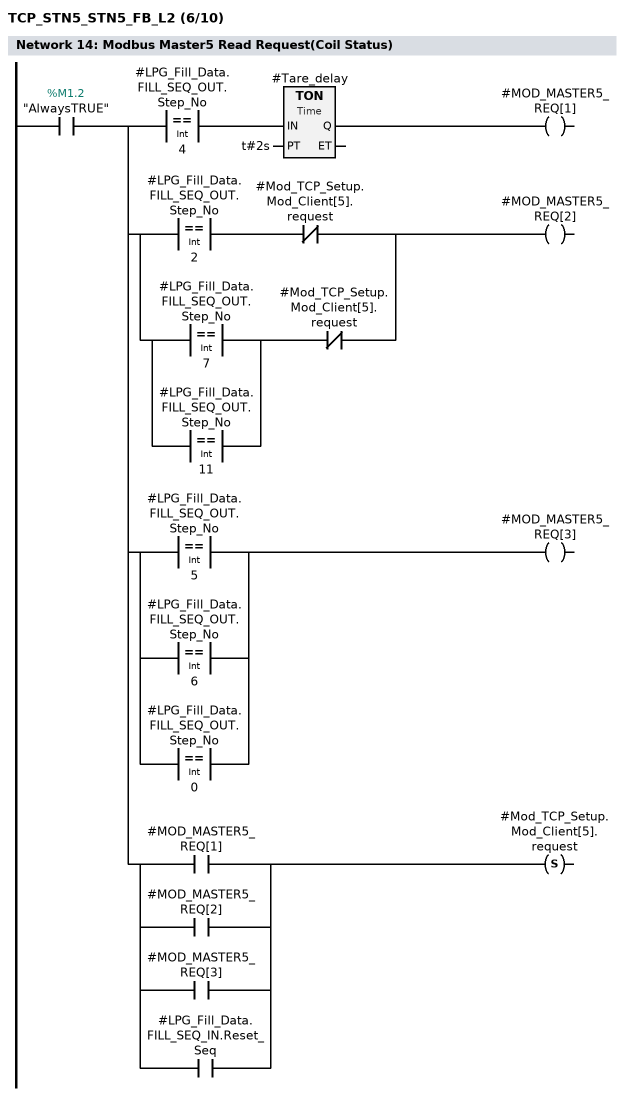
   RUNG wire#powerrail
      Contact( "AlwaysTRUE" )
      wire#w1
      { S7_Templates := "SrcType := Int" } EQ_Contact(in1 := #LPG_Fill_Data.FILL_SEQ_OUT.Step_No, in2 := 4)
      { S7_Templates := "time_type := Time" } #Tare_delay.TON(pt := t#2s, et =>)
      Coil( #MOD_MASTER5_REQ[1] )
   END_RUNG
   RUNG wire#w1
      { S7_Templates := "SrcType := Int" } EQ_Contact(in1 := #LPG_Fill_Data.FILL_SEQ_OUT.Step_No, in2 := 2)
      I_Contact( #Mod_TCP_Setup.Mod_Client[5].request )
      wire#w2
      Coil( #MOD_MASTER5_REQ[2] )
   END_RUNG
   RUNG wire#w1
      { S7_Templates := "SrcType := Int" } EQ_Contact(in1 := #LPG_Fill_Data.FILL_SEQ_OUT.Step_No, in2 := 7)
      wire#w3
      I_Contact( #Mod_TCP_Setup.Mod_Client[5].request )
   END_RUNG wire#w2
   RUNG wire#w1
      { S7_Templates := "SrcType := Int" } EQ_Contact(in1 := #LPG_Fill_Data.FILL_SEQ_OUT.Step_No, in2 := 11)
   END_RUNG wire#w3
   RUNG wire#w1
      { S7_Templates := "SrcType := Int" } EQ_Contact(in1 := #LPG_Fill_Data.FILL_SEQ_OUT.Step_No, in2 := 5)
      wire#w4
      Coil( #MOD_MASTER5_REQ[3] )
   END_RUNG
   RUNG wire#w1
      { S7_Templates := "SrcType := Int" } EQ_Contact(in1 := #LPG_Fill_Data.FILL_SEQ_OUT.Step_No, in2 := 6)
   END_RUNG wire#w4
   RUNG wire#w1
      { S7_Templates := "SrcType := Int" } EQ_Contact(in1 := #LPG_Fill_Data.FILL_SEQ_OUT.Step_No, in2 := 0)
   END_RUNG wire#w4
   RUNG wire#w1
      Contact( #MOD_MASTER5_REQ[1] )
      wire#w5
      S_Coil( #Mod_TCP_Setup.Mod_Client[5].request )
   END_RUNG
   RUNG wire#w1
      Contact( #MOD_MASTER5_REQ[2] )
   END_RUNG wire#w5
   RUNG wire#w1
      Contact( #MOD_MASTER5_REQ[3] )
   END_RUNG wire#w5
   RUNG wire#w1
      Contact( #LPG_Fill_Data.FILL_SEQ_IN.Reset_Seq )
   END_RUNG wire#w5
   // the same network as SCL:
   #Tare_delay(IN := "AlwaysTRUE" AND (#LPG_Fill_Data.FILL_SEQ_OUT.Step_No = 4), PT := t#2s);   // TON
   #MOD_MASTER5_REQ[1] := #Tare_delay.Q;
   #MOD_MASTER5_REQ[2] := "AlwaysTRUE" AND (((#LPG_Fill_Data.FILL_SEQ_OUT.Step_No = 2) AND NOT #Mod_TCP_Setup.Mod_Client[5].request) OR (((#LPG_Fill_Data.FILL_SEQ_OUT.Step_No = 7) OR (#LPG_Fill_Data.FILL_SEQ_OUT.Step_No = 11)) AND NOT #Mod_TCP_Setup.Mod_Client[5].request));
   #MOD_MASTER5_REQ[3] := "AlwaysTRUE" AND ((#LPG_Fill_Data.FILL_SEQ_OUT.Step_No = 5) OR (#LPG_Fill_Data.FILL_SEQ_OUT.Step_No = 6) OR (#LPG_Fill_Data.FILL_SEQ_OUT.Step_No = 0));
   IF "AlwaysTRUE" AND (#MOD_MASTER5_REQ[1] OR #MOD_MASTER5_REQ[2] OR #MOD_MASTER5_REQ[3] OR #LPG_Fill_Data.FILL_SEQ_IN.Reset_Seq) THEN
       #Mod_TCP_Setup.Mod_Client[5].request := TRUE;
   END_IF;
END_REGION

REGION Network 15: Modbus Master5 Read Coil Status
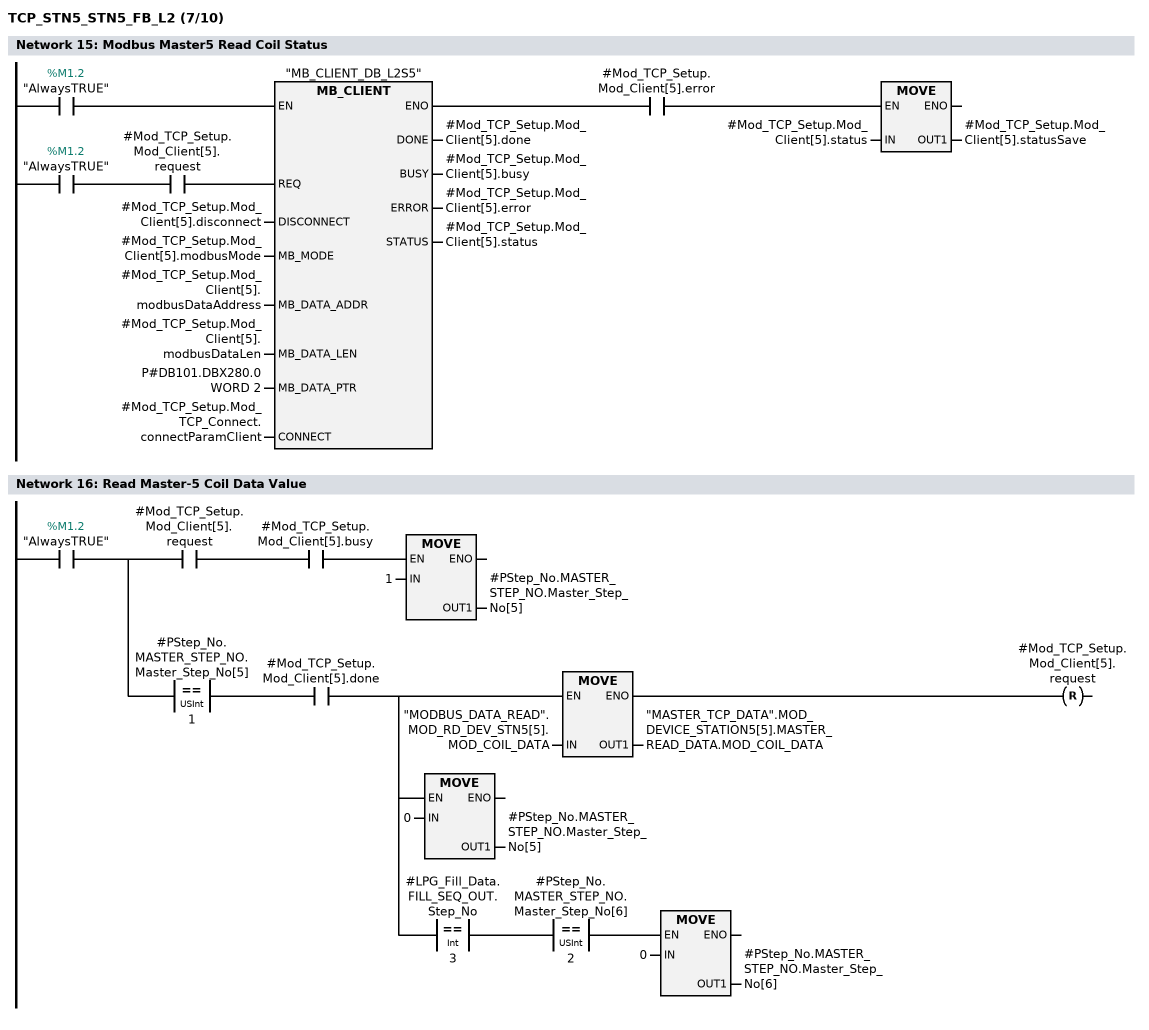
   RUNG wire#powerrail
      Contact( "AlwaysTRUE" )
      "MB_CLIENT_DB_L2S5".MB_CLIENT(REQ := wire#w1, DISCONNECT := #Mod_TCP_Setup.Mod_Client[5].disconnect, MB_MODE := #Mod_TCP_Setup.Mod_Client[5].modbusMode, MB_DATA_ADDR := #Mod_TCP_Setup.Mod_Client[5].modbusDataAddress, MB_DATA_LEN := #Mod_TCP_Setup.Mod_Client[5].modbusDataLen, MB_DATA_PTR := P#DB101.DBX280.0 WORD 2, CONNECT := #Mod_TCP_Setup.Mod_TCP_Connect.connectParamClient, DONE => #Mod_TCP_Setup.Mod_Client[5].done, BUSY => #Mod_TCP_Setup.Mod_Client[5].busy, ERROR => #Mod_TCP_Setup.Mod_Client[5].error, STATUS => #Mod_TCP_Setup.Mod_Client[5].status)
      Contact( #Mod_TCP_Setup.Mod_Client[5].error )
      Move(in := #Mod_TCP_Setup.Mod_Client[5].status, out1 => #Mod_TCP_Setup.Mod_Client[5].statusSave)
   END_RUNG
   RUNG wire#powerrail
      Contact( "AlwaysTRUE" )
      Contact( #Mod_TCP_Setup.Mod_Client[5].request )
   END_RUNG wire#w1
   // the same network as SCL:
   "MB_CLIENT_DB_L2S5"(EN := "AlwaysTRUE",   // MB_CLIENT
                       REQ := "AlwaysTRUE" AND #Mod_TCP_Setup.Mod_Client[5].request,
                       DISCONNECT := #Mod_TCP_Setup.Mod_Client[5].disconnect,
                       MB_MODE := #Mod_TCP_Setup.Mod_Client[5].modbusMode,
                       MB_DATA_ADDR := #Mod_TCP_Setup.Mod_Client[5].modbusDataAddress,
                       MB_DATA_LEN := #Mod_TCP_Setup.Mod_Client[5].modbusDataLen,
                       MB_DATA_PTR := P#DB101.DBX280.0 WORD 2,
                       CONNECT := #Mod_TCP_Setup.Mod_TCP_Connect.connectParamClient,
                       DONE => #Mod_TCP_Setup.Mod_Client[5].done,
                       BUSY => #Mod_TCP_Setup.Mod_Client[5].busy,
                       ERROR => #Mod_TCP_Setup.Mod_Client[5].error,
                       STATUS => #Mod_TCP_Setup.Mod_Client[5].status,
                       ENO => #_w1);
   IF #_w1 AND #Mod_TCP_Setup.Mod_Client[5].error THEN
       #Mod_TCP_Setup.Mod_Client[5].statusSave := #Mod_TCP_Setup.Mod_Client[5].status;
   END_IF;
END_REGION

REGION Network 16: Read Master-5 Coil Data Value
   RUNG wire#powerrail
      Contact( "AlwaysTRUE" )
      wire#w1
      Contact( #Mod_TCP_Setup.Mod_Client[5].request )
      Contact( #Mod_TCP_Setup.Mod_Client[5].busy )
      Move(in := 1, out1 => #PStep_No.MASTER_STEP_NO.Master_Step_No[5])
   END_RUNG
   RUNG wire#w1
      { S7_Templates := "SrcType := USInt" } EQ_Contact(in1 := #PStep_No.MASTER_STEP_NO.Master_Step_No[5], in2 := 1)
      Contact( #Mod_TCP_Setup.Mod_Client[5].done )
      wire#w2
      Move(in := "MODBUS_DATA_READ".MOD_RD_DEV_STN5[5].MOD_COIL_DATA, out1 => "MASTER_TCP_DATA".MOD_DEVICE_STATION5[5].MASTER_READ_DATA.MOD_COIL_DATA)
      R_Coil( #Mod_TCP_Setup.Mod_Client[5].request )
   END_RUNG
   RUNG wire#w2
      Move(in := 0, out1 => #PStep_No.MASTER_STEP_NO.Master_Step_No[5])
   END_RUNG
   RUNG wire#w2
      { S7_Templates := "SrcType := Int" } EQ_Contact(in1 := #LPG_Fill_Data.FILL_SEQ_OUT.Step_No, in2 := 3)
      { S7_Templates := "SrcType := USInt" } EQ_Contact(in1 := #PStep_No.MASTER_STEP_NO.Master_Step_No[6], in2 := 2)
      Move(in := 0, out1 => #PStep_No.MASTER_STEP_NO.Master_Step_No[6])
   END_RUNG
   // the same network as SCL:
   IF "AlwaysTRUE" AND #Mod_TCP_Setup.Mod_Client[5].request AND #Mod_TCP_Setup.Mod_Client[5].busy THEN
       #PStep_No.MASTER_STEP_NO.Master_Step_No[5] := 1;
   END_IF;
   #_w1 := "AlwaysTRUE" AND (#PStep_No.MASTER_STEP_NO.Master_Step_No[5] = 1) AND #Mod_TCP_Setup.Mod_Client[5].done;
   IF #_w1 THEN
       "MASTER_TCP_DATA".MOD_DEVICE_STATION5[5].MASTER_READ_DATA.MOD_COIL_DATA := "MODBUS_DATA_READ".MOD_RD_DEV_STN5[5].MOD_COIL_DATA;
       #Mod_TCP_Setup.Mod_Client[5].request := FALSE;
       #PStep_No.MASTER_STEP_NO.Master_Step_No[5] := 0;
   END_IF;
   IF #_w1 AND (#LPG_Fill_Data.FILL_SEQ_OUT.Step_No = 3) AND (#PStep_No.MASTER_STEP_NO.Master_Step_No[6] = 2) THEN
       #PStep_No.MASTER_STEP_NO.Master_Step_No[6] := 0;
   END_IF;
END_REGION

REGION Network 17: Write Coil Data
   // if multiple bit write not working
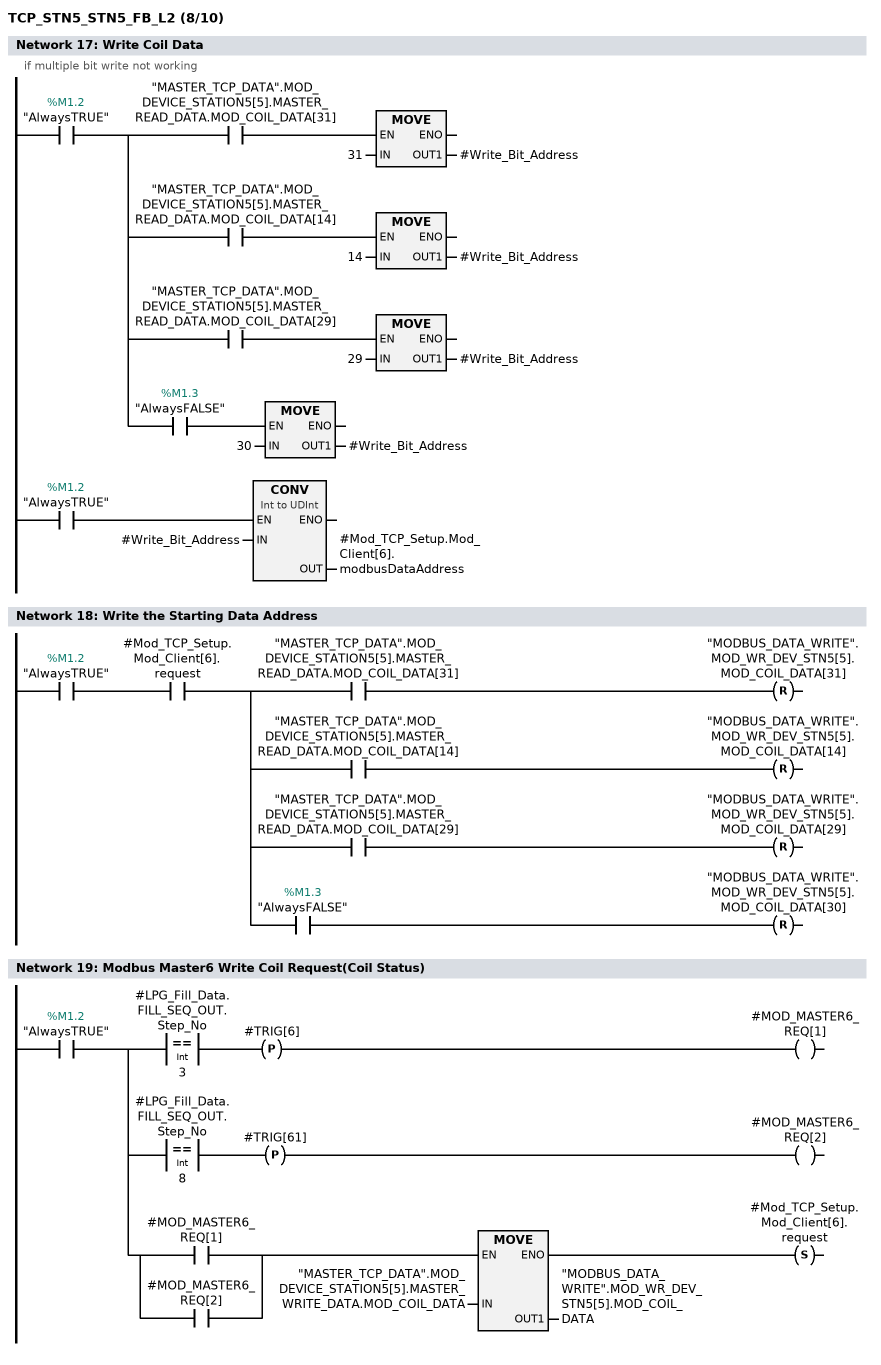
   RUNG wire#powerrail
      Contact( "AlwaysTRUE" )
      wire#w1
      Contact( "MASTER_TCP_DATA".MOD_DEVICE_STATION5[5].MASTER_READ_DATA.MOD_COIL_DATA[31] )
      Move(in := 31, out1 => #Write_Bit_Address)
   END_RUNG
   RUNG wire#w1
      Contact( "MASTER_TCP_DATA".MOD_DEVICE_STATION5[5].MASTER_READ_DATA.MOD_COIL_DATA[14] )
      Move(in := 14, out1 => #Write_Bit_Address)
   END_RUNG
   RUNG wire#w1
      Contact( "MASTER_TCP_DATA".MOD_DEVICE_STATION5[5].MASTER_READ_DATA.MOD_COIL_DATA[29] )
      Move(in := 29, out1 => #Write_Bit_Address)
   END_RUNG
   RUNG wire#w1
      Contact( "AlwaysFALSE" )
      Move(in := 30, out1 => #Write_Bit_Address)
   END_RUNG
   RUNG wire#powerrail
      Contact( "AlwaysTRUE" )
      { S7_Templates := "[SrcType := Int, DestType := UDInt]" } Convert(in := #Write_Bit_Address, out => #Mod_TCP_Setup.Mod_Client[6].modbusDataAddress)
   END_RUNG
   // the same network as SCL:
   IF "AlwaysTRUE" AND "MASTER_TCP_DATA".MOD_DEVICE_STATION5[5].MASTER_READ_DATA.MOD_COIL_DATA[31] THEN
       #Write_Bit_Address := 31;
   END_IF;
   IF "AlwaysTRUE" AND "MASTER_TCP_DATA".MOD_DEVICE_STATION5[5].MASTER_READ_DATA.MOD_COIL_DATA[14] THEN
       #Write_Bit_Address := 14;
   END_IF;
   IF "AlwaysTRUE" AND "MASTER_TCP_DATA".MOD_DEVICE_STATION5[5].MASTER_READ_DATA.MOD_COIL_DATA[29] THEN
       #Write_Bit_Address := 29;
   END_IF;
   IF "AlwaysTRUE" AND "AlwaysFALSE" THEN #Write_Bit_Address := 30; END_IF;
   IF "AlwaysTRUE" THEN
       #Mod_TCP_Setup.Mod_Client[6].modbusDataAddress := INT_TO_UDINT(#Write_Bit_Address);
   END_IF;
END_REGION

REGION Network 18: Write the Starting Data Address
   RUNG wire#powerrail
      Contact( "AlwaysTRUE" )
      Contact( #Mod_TCP_Setup.Mod_Client[6].request )
      wire#w1
      Contact( "MASTER_TCP_DATA".MOD_DEVICE_STATION5[5].MASTER_READ_DATA.MOD_COIL_DATA[31] )
      R_Coil( "MODBUS_DATA_WRITE".MOD_WR_DEV_STN5[5].MOD_COIL_DATA[31] )
   END_RUNG
   RUNG wire#w1
      Contact( "MASTER_TCP_DATA".MOD_DEVICE_STATION5[5].MASTER_READ_DATA.MOD_COIL_DATA[14] )
      R_Coil( "MODBUS_DATA_WRITE".MOD_WR_DEV_STN5[5].MOD_COIL_DATA[14] )
   END_RUNG
   RUNG wire#w1
      Contact( "MASTER_TCP_DATA".MOD_DEVICE_STATION5[5].MASTER_READ_DATA.MOD_COIL_DATA[29] )
      R_Coil( "MODBUS_DATA_WRITE".MOD_WR_DEV_STN5[5].MOD_COIL_DATA[29] )
   END_RUNG
   RUNG wire#w1
      Contact( "AlwaysFALSE" )
      R_Coil( "MODBUS_DATA_WRITE".MOD_WR_DEV_STN5[5].MOD_COIL_DATA[30] )
   END_RUNG
   // the same network as SCL:
   #_w1 := "AlwaysTRUE" AND #Mod_TCP_Setup.Mod_Client[6].request;
   IF #_w1 AND "MASTER_TCP_DATA".MOD_DEVICE_STATION5[5].MASTER_READ_DATA.MOD_COIL_DATA[31] THEN
       "MODBUS_DATA_WRITE".MOD_WR_DEV_STN5[5].MOD_COIL_DATA[31] := FALSE;
   END_IF;
   IF #_w1 AND "MASTER_TCP_DATA".MOD_DEVICE_STATION5[5].MASTER_READ_DATA.MOD_COIL_DATA[14] THEN
       "MODBUS_DATA_WRITE".MOD_WR_DEV_STN5[5].MOD_COIL_DATA[14] := FALSE;
   END_IF;
   IF #_w1 AND "MASTER_TCP_DATA".MOD_DEVICE_STATION5[5].MASTER_READ_DATA.MOD_COIL_DATA[29] THEN
       "MODBUS_DATA_WRITE".MOD_WR_DEV_STN5[5].MOD_COIL_DATA[29] := FALSE;
   END_IF;
   IF #_w1 AND "AlwaysFALSE" THEN "MODBUS_DATA_WRITE".MOD_WR_DEV_STN5[5].MOD_COIL_DATA[30] := FALSE; END_IF;
END_REGION

REGION Network 19: Modbus Master6 Write Coil Request(Coil Status)
   RUNG wire#powerrail
      Contact( "AlwaysTRUE" )
      wire#w1
      { S7_Templates := "SrcType := Int" } EQ_Contact(in1 := #LPG_Fill_Data.FILL_SEQ_OUT.Step_No, in2 := 3)
      P_Trig( #TRIG[6] )
      Coil( #MOD_MASTER6_REQ[1] )
   END_RUNG
   RUNG wire#w1
      { S7_Templates := "SrcType := Int" } EQ_Contact(in1 := #LPG_Fill_Data.FILL_SEQ_OUT.Step_No, in2 := 8)
      P_Trig( #TRIG[61] )
      Coil( #MOD_MASTER6_REQ[2] )
   END_RUNG
   RUNG wire#w1
      Contact( #MOD_MASTER6_REQ[1] )
      wire#w2
      Move(in := "MASTER_TCP_DATA".MOD_DEVICE_STATION5[5].MASTER_WRITE_DATA.MOD_COIL_DATA, out1 => "MODBUS_DATA_WRITE".MOD_WR_DEV_STN5[5].MOD_COIL_DATA)
      S_Coil( #Mod_TCP_Setup.Mod_Client[6].request )
   END_RUNG
   RUNG wire#w1
      Contact( #MOD_MASTER6_REQ[2] )
   END_RUNG wire#w2
   // the same network as SCL:
   #_w1 := "AlwaysTRUE" AND (#LPG_Fill_Data.FILL_SEQ_OUT.Step_No = 3);
   #_w2 := #_w1 AND NOT #TRIG[6];   // rising edge
   #TRIG[6] := #_w1;
   #MOD_MASTER6_REQ[1] := #_w2;
   #_w3 := "AlwaysTRUE" AND (#LPG_Fill_Data.FILL_SEQ_OUT.Step_No = 8);
   #_w4 := #_w3 AND NOT #TRIG[61];   // rising edge
   #TRIG[61] := #_w3;
   #MOD_MASTER6_REQ[2] := #_w4;
   IF "AlwaysTRUE" AND (#MOD_MASTER6_REQ[1] OR #MOD_MASTER6_REQ[2]) THEN
       "MODBUS_DATA_WRITE".MOD_WR_DEV_STN5[5].MOD_COIL_DATA := "MASTER_TCP_DATA".MOD_DEVICE_STATION5[5].MASTER_WRITE_DATA.MOD_COIL_DATA;
       #Mod_TCP_Setup.Mod_Client[6].request := TRUE;
   END_IF;
END_REGION

REGION Network 20: Modbus Master6 Write Coil Status
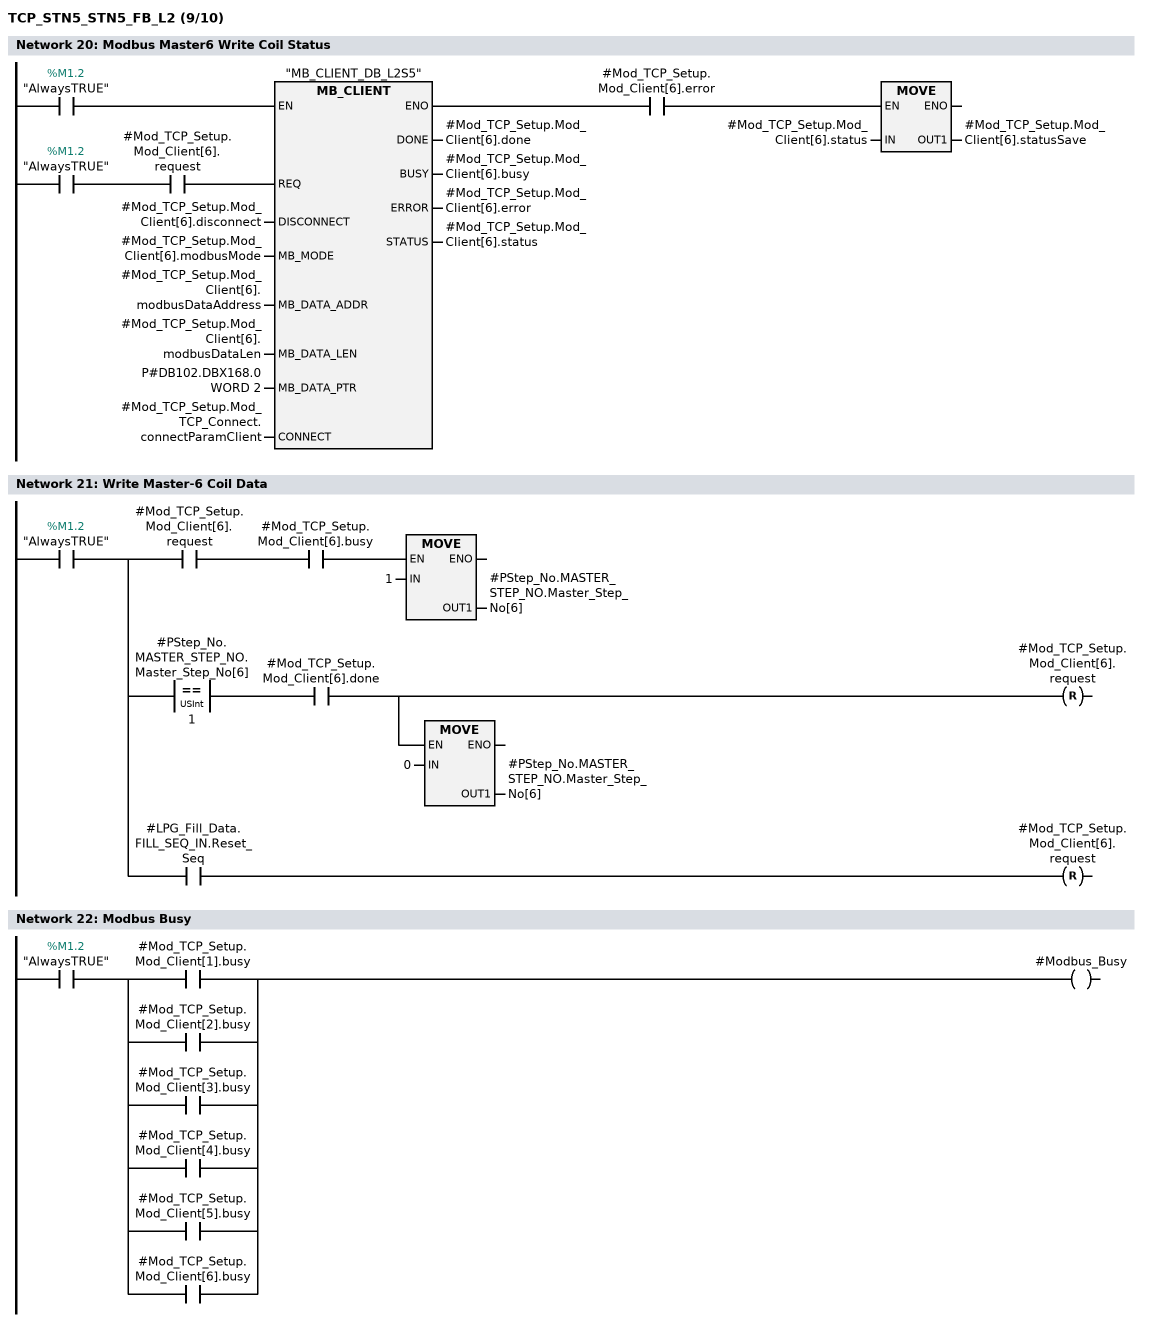
   RUNG wire#powerrail
      Contact( "AlwaysTRUE" )
      "MB_CLIENT_DB_L2S5".MB_CLIENT(REQ := wire#w1, DISCONNECT := #Mod_TCP_Setup.Mod_Client[6].disconnect, MB_MODE := #Mod_TCP_Setup.Mod_Client[6].modbusMode, MB_DATA_ADDR := #Mod_TCP_Setup.Mod_Client[6].modbusDataAddress, MB_DATA_LEN := #Mod_TCP_Setup.Mod_Client[6].modbusDataLen, MB_DATA_PTR := P#DB102.DBX168.0 WORD 2, CONNECT := #Mod_TCP_Setup.Mod_TCP_Connect.connectParamClient, DONE => #Mod_TCP_Setup.Mod_Client[6].done, BUSY => #Mod_TCP_Setup.Mod_Client[6].busy, ERROR => #Mod_TCP_Setup.Mod_Client[6].error, STATUS => #Mod_TCP_Setup.Mod_Client[6].status)
      Contact( #Mod_TCP_Setup.Mod_Client[6].error )
      Move(in := #Mod_TCP_Setup.Mod_Client[6].status, out1 => #Mod_TCP_Setup.Mod_Client[6].statusSave)
   END_RUNG
   RUNG wire#powerrail
      Contact( "AlwaysTRUE" )
      Contact( #Mod_TCP_Setup.Mod_Client[6].request )
   END_RUNG wire#w1
   // the same network as SCL:
   "MB_CLIENT_DB_L2S5"(EN := "AlwaysTRUE",   // MB_CLIENT
                       REQ := "AlwaysTRUE" AND #Mod_TCP_Setup.Mod_Client[6].request,
                       DISCONNECT := #Mod_TCP_Setup.Mod_Client[6].disconnect,
                       MB_MODE := #Mod_TCP_Setup.Mod_Client[6].modbusMode,
                       MB_DATA_ADDR := #Mod_TCP_Setup.Mod_Client[6].modbusDataAddress,
                       MB_DATA_LEN := #Mod_TCP_Setup.Mod_Client[6].modbusDataLen,
                       MB_DATA_PTR := P#DB102.DBX168.0 WORD 2,
                       CONNECT := #Mod_TCP_Setup.Mod_TCP_Connect.connectParamClient,
                       DONE => #Mod_TCP_Setup.Mod_Client[6].done,
                       BUSY => #Mod_TCP_Setup.Mod_Client[6].busy,
                       ERROR => #Mod_TCP_Setup.Mod_Client[6].error,
                       STATUS => #Mod_TCP_Setup.Mod_Client[6].status,
                       ENO => #_w1);
   IF #_w1 AND #Mod_TCP_Setup.Mod_Client[6].error THEN
       #Mod_TCP_Setup.Mod_Client[6].statusSave := #Mod_TCP_Setup.Mod_Client[6].status;
   END_IF;
END_REGION

REGION Network 21: Write Master-6 Coil Data
   RUNG wire#powerrail
      Contact( "AlwaysTRUE" )
      wire#w1
      Contact( #Mod_TCP_Setup.Mod_Client[6].request )
      Contact( #Mod_TCP_Setup.Mod_Client[6].busy )
      Move(in := 1, out1 => #PStep_No.MASTER_STEP_NO.Master_Step_No[6])
   END_RUNG
   RUNG wire#w1
      { S7_Templates := "SrcType := USInt" } EQ_Contact(in1 := #PStep_No.MASTER_STEP_NO.Master_Step_No[6], in2 := 1)
      Contact( #Mod_TCP_Setup.Mod_Client[6].done )
      wire#w2
      R_Coil( #Mod_TCP_Setup.Mod_Client[6].request )
   END_RUNG
   RUNG wire#w2
      Move(in := 0, out1 => #PStep_No.MASTER_STEP_NO.Master_Step_No[6])
   END_RUNG
   RUNG wire#w1
      Contact( #LPG_Fill_Data.FILL_SEQ_IN.Reset_Seq )
      R_Coil( #Mod_TCP_Setup.Mod_Client[6].request )
   END_RUNG
   // the same network as SCL:
   IF "AlwaysTRUE" AND #Mod_TCP_Setup.Mod_Client[6].request AND #Mod_TCP_Setup.Mod_Client[6].busy THEN
       #PStep_No.MASTER_STEP_NO.Master_Step_No[6] := 1;
   END_IF;
   #_w1 := "AlwaysTRUE" AND (#PStep_No.MASTER_STEP_NO.Master_Step_No[6] = 1) AND #Mod_TCP_Setup.Mod_Client[6].done;
   IF #_w1 THEN
       #Mod_TCP_Setup.Mod_Client[6].request := FALSE;
       #PStep_No.MASTER_STEP_NO.Master_Step_No[6] := 0;
   END_IF;
   IF "AlwaysTRUE" AND #LPG_Fill_Data.FILL_SEQ_IN.Reset_Seq THEN
       #Mod_TCP_Setup.Mod_Client[6].request := FALSE;
   END_IF;
END_REGION

REGION Network 22: Modbus Busy
   RUNG wire#powerrail
      Contact( "AlwaysTRUE" )
      wire#w1
      Contact( #Mod_TCP_Setup.Mod_Client[1].busy )
      wire#w2
      Coil( #Modbus_Busy )
   END_RUNG
   RUNG wire#w1
      Contact( #Mod_TCP_Setup.Mod_Client[2].busy )
   END_RUNG wire#w2
   RUNG wire#w1
      Contact( #Mod_TCP_Setup.Mod_Client[3].busy )
   END_RUNG wire#w2
   RUNG wire#w1
      Contact( #Mod_TCP_Setup.Mod_Client[4].busy )
   END_RUNG wire#w2
   RUNG wire#w1
      Contact( #Mod_TCP_Setup.Mod_Client[5].busy )
   END_RUNG wire#w2
   RUNG wire#w1
      Contact( #Mod_TCP_Setup.Mod_Client[6].busy )
   END_RUNG wire#w2
   // the same network as SCL:
   #Modbus_Busy := "AlwaysTRUE" AND (#Mod_TCP_Setup.Mod_Client[1].busy OR #Mod_TCP_Setup.Mod_Client[2].busy OR #Mod_TCP_Setup.Mod_Client[3].busy OR #Mod_TCP_Setup.Mod_Client[4].busy OR #Mod_TCP_Setup.Mod_Client[5].busy OR #Mod_TCP_Setup.Mod_Client[6].busy);
END_REGION

REGION Network 23
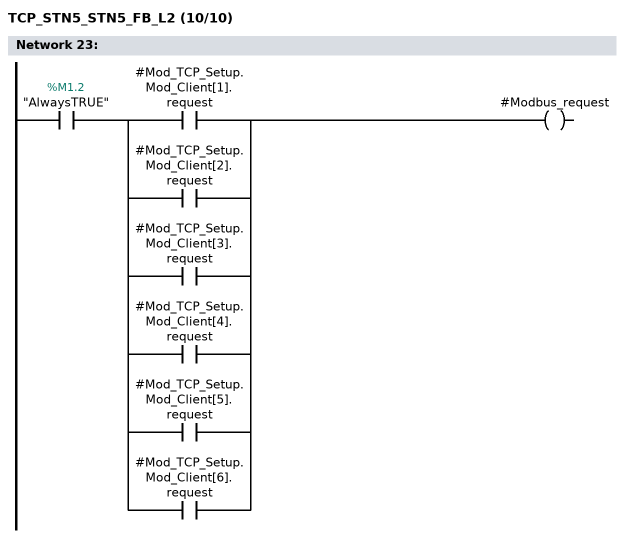
   RUNG wire#powerrail
      Contact( "AlwaysTRUE" )
      wire#w1
      Contact( #Mod_TCP_Setup.Mod_Client[1].request )
      wire#w2
      Coil( #Modbus_request )
   END_RUNG
   RUNG wire#w1
      Contact( #Mod_TCP_Setup.Mod_Client[2].request )
   END_RUNG wire#w2
   RUNG wire#w1
      Contact( #Mod_TCP_Setup.Mod_Client[3].request )
   END_RUNG wire#w2
   RUNG wire#w1
      Contact( #Mod_TCP_Setup.Mod_Client[4].request )
   END_RUNG wire#w2
   RUNG wire#w1
      Contact( #Mod_TCP_Setup.Mod_Client[5].request )
   END_RUNG wire#w2
   RUNG wire#w1
      Contact( #Mod_TCP_Setup.Mod_Client[6].request )
   END_RUNG wire#w2
   // the same network as SCL:
   #Modbus_request := "AlwaysTRUE" AND (#Mod_TCP_Setup.Mod_Client[1].request OR #Mod_TCP_Setup.Mod_Client[2].request OR #Mod_TCP_Setup.Mod_Client[3].request OR #Mod_TCP_Setup.Mod_Client[4].request OR #Mod_TCP_Setup.Mod_Client[5].request OR #Mod_TCP_Setup.Mod_Client[6].request);
END_REGION
END_FUNCTION_BLOCK

FUNCTION_BLOCK "TCP_STN5_STN6_FB_L2"   // FB260, LAD
{ S7_Optimized_Access := 'TRUE' }
VERSION : 0.1
// stored: AutoNumber false, IsIECCheckEnabled false, IsRetainMemResEnabled false, MemoryReserve 100, SetENOAutomatically false, UDAEnableTagReadback false
   VAR_OUTPUT
      Modbus_Busy : Bool;
   END_VAR
   VAR_IN_OUT
      Mod_TCP_Setup : "Mod_TCP_Data";
      LPG_Fill_Data : "LPG_FILL_DATA";
   END_VAR
   VAR
      PStep_No : Struct
         MASTER_STEP_NO : "Master_Step_No";
      END_STRUCT;
      Write_Bit_Address : Int;
      TRIG : Array[1..100] of Bool;
      MOD_MASTER1_REQ : Array[1..10] of Bool;
      MOD_MASTER2_REQ : Array[1..10] of Bool;
      MOD_MASTER3_REQ : Array[1..10] of Bool;
      MOD_MASTER4_REQ : Array[1..10] of Bool;
      MOD_MASTER5_REQ : Array[1..10] of Bool;
      MOD_MASTER6_REQ : Array[1..10] of Bool;
      MAS_TRG_EXTN { S7_SetPoint := 'True'} : TOF_TIME;
      Tare_delay { S7_SetPoint := 'True'} : TON_TIME;
   END_VAR
   VAR_TEMP
      Modbus_request : Bool;
   END_VAR
   VAR_TEMP   // added for the SCL form of the ladder/FBD networks
      _w1 : Bool;
      _w2 : Bool;
      _w3 : Bool;
      _w4 : Bool;
      _w5 : Bool;
      _w6 : Bool;
   END_VAR
BEGIN

REGION Network 1: FILLING LINE-1 STATION-6
END_REGION

REGION Network 2: Write Master-1 Holding Register Request(Tare Weight Entry)
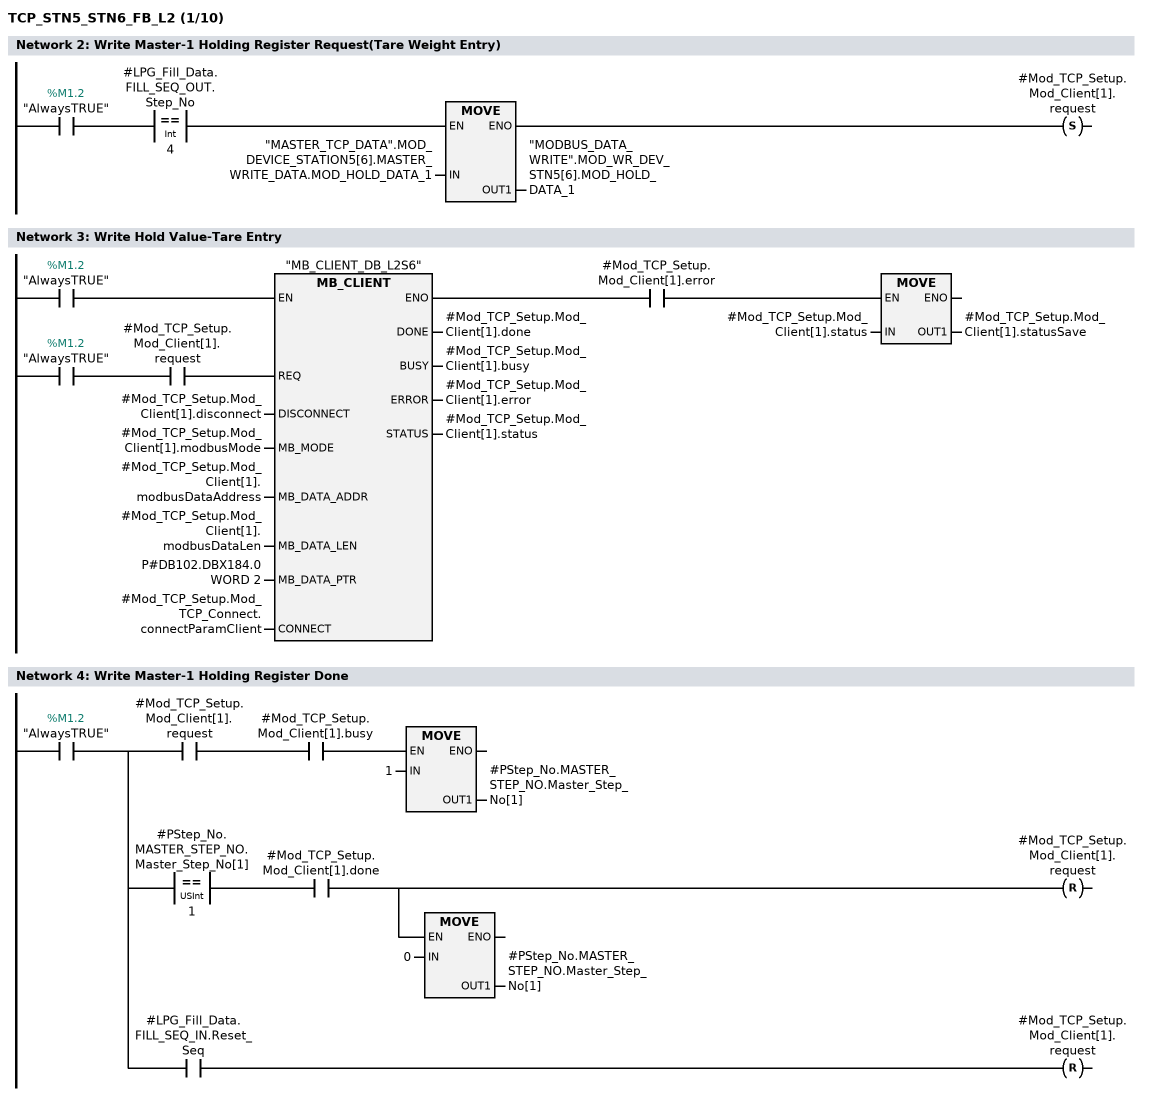
   RUNG wire#powerrail
      Contact( "AlwaysTRUE" )
      { S7_Templates := "SrcType := Int" } EQ_Contact(in1 := #LPG_Fill_Data.FILL_SEQ_OUT.Step_No, in2 := 4)
      Move(in := "MASTER_TCP_DATA".MOD_DEVICE_STATION5[6].MASTER_WRITE_DATA.MOD_HOLD_DATA_1, out1 => "MODBUS_DATA_WRITE".MOD_WR_DEV_STN5[6].MOD_HOLD_DATA_1)
      S_Coil( #Mod_TCP_Setup.Mod_Client[1].request )
   END_RUNG
   // the same network as SCL:
   IF "AlwaysTRUE" AND (#LPG_Fill_Data.FILL_SEQ_OUT.Step_No = 4) THEN
       "MODBUS_DATA_WRITE".MOD_WR_DEV_STN5[6].MOD_HOLD_DATA_1 := "MASTER_TCP_DATA".MOD_DEVICE_STATION5[6].MASTER_WRITE_DATA.MOD_HOLD_DATA_1;
       #Mod_TCP_Setup.Mod_Client[1].request := TRUE;
   END_IF;
END_REGION

REGION Network 3: Write Hold Value-Tare Entry
   RUNG wire#powerrail
      Contact( "AlwaysTRUE" )
      "MB_CLIENT_DB_L2S6".MB_CLIENT(REQ := wire#w1, DISCONNECT := #Mod_TCP_Setup.Mod_Client[1].disconnect, MB_MODE := #Mod_TCP_Setup.Mod_Client[1].modbusMode, MB_DATA_ADDR := #Mod_TCP_Setup.Mod_Client[1].modbusDataAddress, MB_DATA_LEN := #Mod_TCP_Setup.Mod_Client[1].modbusDataLen, MB_DATA_PTR := P#DB102.DBX184.0 WORD 2, CONNECT := #Mod_TCP_Setup.Mod_TCP_Connect.connectParamClient, DONE => #Mod_TCP_Setup.Mod_Client[1].done, BUSY => #Mod_TCP_Setup.Mod_Client[1].busy, ERROR => #Mod_TCP_Setup.Mod_Client[1].error, STATUS => #Mod_TCP_Setup.Mod_Client[1].status)
      Contact( #Mod_TCP_Setup.Mod_Client[1].error )
      Move(in := #Mod_TCP_Setup.Mod_Client[1].status, out1 => #Mod_TCP_Setup.Mod_Client[1].statusSave)
   END_RUNG
   RUNG wire#powerrail
      Contact( "AlwaysTRUE" )
      Contact( #Mod_TCP_Setup.Mod_Client[1].request )
   END_RUNG wire#w1
   // the same network as SCL:
   "MB_CLIENT_DB_L2S6"(EN := "AlwaysTRUE",   // MB_CLIENT
                       REQ := "AlwaysTRUE" AND #Mod_TCP_Setup.Mod_Client[1].request,
                       DISCONNECT := #Mod_TCP_Setup.Mod_Client[1].disconnect,
                       MB_MODE := #Mod_TCP_Setup.Mod_Client[1].modbusMode,
                       MB_DATA_ADDR := #Mod_TCP_Setup.Mod_Client[1].modbusDataAddress,
                       MB_DATA_LEN := #Mod_TCP_Setup.Mod_Client[1].modbusDataLen,
                       MB_DATA_PTR := P#DB102.DBX184.0 WORD 2,
                       CONNECT := #Mod_TCP_Setup.Mod_TCP_Connect.connectParamClient,
                       DONE => #Mod_TCP_Setup.Mod_Client[1].done,
                       BUSY => #Mod_TCP_Setup.Mod_Client[1].busy,
                       ERROR => #Mod_TCP_Setup.Mod_Client[1].error,
                       STATUS => #Mod_TCP_Setup.Mod_Client[1].status,
                       ENO => #_w1);
   IF #_w1 AND #Mod_TCP_Setup.Mod_Client[1].error THEN
       #Mod_TCP_Setup.Mod_Client[1].statusSave := #Mod_TCP_Setup.Mod_Client[1].status;
   END_IF;
END_REGION

REGION Network 4: Write Master-1 Holding Register Done
   RUNG wire#powerrail
      Contact( "AlwaysTRUE" )
      wire#w1
      Contact( #Mod_TCP_Setup.Mod_Client[1].request )
      Contact( #Mod_TCP_Setup.Mod_Client[1].busy )
      Move(in := 1, out1 => #PStep_No.MASTER_STEP_NO.Master_Step_No[1])
   END_RUNG
   RUNG wire#w1
      { S7_Templates := "SrcType := USInt" } EQ_Contact(in1 := #PStep_No.MASTER_STEP_NO.Master_Step_No[1], in2 := 1)
      Contact( #Mod_TCP_Setup.Mod_Client[1].done )
      wire#w2
      R_Coil( #Mod_TCP_Setup.Mod_Client[1].request )
   END_RUNG
   RUNG wire#w2
      Move(in := 0, out1 => #PStep_No.MASTER_STEP_NO.Master_Step_No[1])
   END_RUNG
   RUNG wire#w1
      Contact( #LPG_Fill_Data.FILL_SEQ_IN.Reset_Seq )
      R_Coil( #Mod_TCP_Setup.Mod_Client[1].request )
   END_RUNG
   // the same network as SCL:
   IF "AlwaysTRUE" AND #Mod_TCP_Setup.Mod_Client[1].request AND #Mod_TCP_Setup.Mod_Client[1].busy THEN
       #PStep_No.MASTER_STEP_NO.Master_Step_No[1] := 1;
   END_IF;
   #_w1 := "AlwaysTRUE" AND (#PStep_No.MASTER_STEP_NO.Master_Step_No[1] = 1) AND #Mod_TCP_Setup.Mod_Client[1].done;
   IF #_w1 THEN
       #Mod_TCP_Setup.Mod_Client[1].request := FALSE;
       #PStep_No.MASTER_STEP_NO.Master_Step_No[1] := 0;
   END_IF;
   IF "AlwaysTRUE" AND #LPG_Fill_Data.FILL_SEQ_IN.Reset_Seq THEN
       #Mod_TCP_Setup.Mod_Client[1].request := FALSE;
   END_IF;
END_REGION

REGION Network 5: Modbus Master2 Read Request(Filled Data)
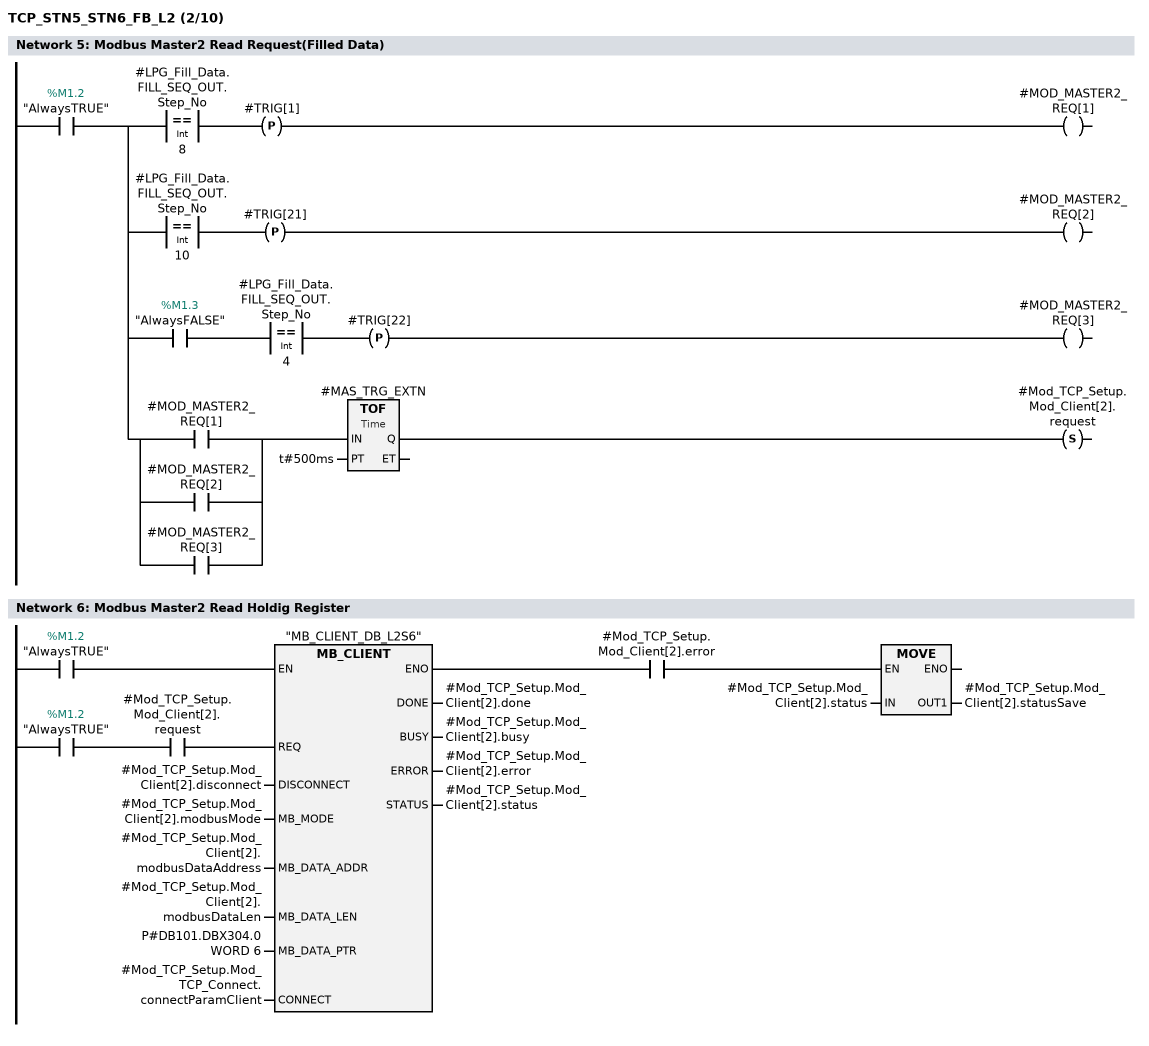
   RUNG wire#powerrail
      Contact( "AlwaysTRUE" )
      wire#w1
      { S7_Templates := "SrcType := Int" } EQ_Contact(in1 := #LPG_Fill_Data.FILL_SEQ_OUT.Step_No, in2 := 8)
      P_Trig( #TRIG[1] )
      Coil( #MOD_MASTER2_REQ[1] )
   END_RUNG
   RUNG wire#w1
      { S7_Templates := "SrcType := Int" } EQ_Contact(in1 := #LPG_Fill_Data.FILL_SEQ_OUT.Step_No, in2 := 10)
      P_Trig( #TRIG[21] )
      Coil( #MOD_MASTER2_REQ[2] )
   END_RUNG
   RUNG wire#w1
      Contact( "AlwaysFALSE" )
      { S7_Templates := "SrcType := Int" } EQ_Contact(in1 := #LPG_Fill_Data.FILL_SEQ_OUT.Step_No, in2 := 4)
      P_Trig( #TRIG[22] )
      Coil( #MOD_MASTER2_REQ[3] )
   END_RUNG
   RUNG wire#w1
      Contact( #MOD_MASTER2_REQ[1] )
      wire#w2
      { S7_Templates := "time_type := Time" } #MAS_TRG_EXTN.TOF(pt := t#500ms, et =>)
      S_Coil( #Mod_TCP_Setup.Mod_Client[2].request )
   END_RUNG
   RUNG wire#w1
      Contact( #MOD_MASTER2_REQ[2] )
   END_RUNG wire#w2
   RUNG wire#w1
      Contact( #MOD_MASTER2_REQ[3] )
   END_RUNG wire#w2
   // the same network as SCL:
   #_w1 := "AlwaysTRUE" AND (#LPG_Fill_Data.FILL_SEQ_OUT.Step_No = 8);
   #_w2 := #_w1 AND NOT #TRIG[1];   // rising edge
   #TRIG[1] := #_w1;
   #MOD_MASTER2_REQ[1] := #_w2;
   #_w3 := "AlwaysTRUE" AND (#LPG_Fill_Data.FILL_SEQ_OUT.Step_No = 10);
   #_w4 := #_w3 AND NOT #TRIG[21];   // rising edge
   #TRIG[21] := #_w3;
   #MOD_MASTER2_REQ[2] := #_w4;
   #_w5 := "AlwaysTRUE" AND "AlwaysFALSE" AND (#LPG_Fill_Data.FILL_SEQ_OUT.Step_No = 4);
   #_w6 := #_w5 AND NOT #TRIG[22];   // rising edge
   #TRIG[22] := #_w5;
   #MOD_MASTER2_REQ[3] := #_w6;
   #MAS_TRG_EXTN(IN := "AlwaysTRUE" AND (#MOD_MASTER2_REQ[1] OR #MOD_MASTER2_REQ[2] OR #MOD_MASTER2_REQ[3]),   // TOF
                 PT := t#500ms);
   IF #MAS_TRG_EXTN.Q THEN #Mod_TCP_Setup.Mod_Client[2].request := TRUE; END_IF;
END_REGION

REGION Network 6: Modbus Master2 Read Holdig Register
   RUNG wire#powerrail
      Contact( "AlwaysTRUE" )
      "MB_CLIENT_DB_L2S6".MB_CLIENT(REQ := wire#w1, DISCONNECT := #Mod_TCP_Setup.Mod_Client[2].disconnect, MB_MODE := #Mod_TCP_Setup.Mod_Client[2].modbusMode, MB_DATA_ADDR := #Mod_TCP_Setup.Mod_Client[2].modbusDataAddress, MB_DATA_LEN := #Mod_TCP_Setup.Mod_Client[2].modbusDataLen, MB_DATA_PTR := P#DB101.DBX304.0 WORD 6, CONNECT := #Mod_TCP_Setup.Mod_TCP_Connect.connectParamClient, DONE => #Mod_TCP_Setup.Mod_Client[2].done, BUSY => #Mod_TCP_Setup.Mod_Client[2].busy, ERROR => #Mod_TCP_Setup.Mod_Client[2].error, STATUS => #Mod_TCP_Setup.Mod_Client[2].status)
      Contact( #Mod_TCP_Setup.Mod_Client[2].error )
      Move(in := #Mod_TCP_Setup.Mod_Client[2].status, out1 => #Mod_TCP_Setup.Mod_Client[2].statusSave)
   END_RUNG
   RUNG wire#powerrail
      Contact( "AlwaysTRUE" )
      Contact( #Mod_TCP_Setup.Mod_Client[2].request )
   END_RUNG wire#w1
   // the same network as SCL:
   "MB_CLIENT_DB_L2S6"(EN := "AlwaysTRUE",   // MB_CLIENT
                       REQ := "AlwaysTRUE" AND #Mod_TCP_Setup.Mod_Client[2].request,
                       DISCONNECT := #Mod_TCP_Setup.Mod_Client[2].disconnect,
                       MB_MODE := #Mod_TCP_Setup.Mod_Client[2].modbusMode,
                       MB_DATA_ADDR := #Mod_TCP_Setup.Mod_Client[2].modbusDataAddress,
                       MB_DATA_LEN := #Mod_TCP_Setup.Mod_Client[2].modbusDataLen,
                       MB_DATA_PTR := P#DB101.DBX304.0 WORD 6,
                       CONNECT := #Mod_TCP_Setup.Mod_TCP_Connect.connectParamClient,
                       DONE => #Mod_TCP_Setup.Mod_Client[2].done,
                       BUSY => #Mod_TCP_Setup.Mod_Client[2].busy,
                       ERROR => #Mod_TCP_Setup.Mod_Client[2].error,
                       STATUS => #Mod_TCP_Setup.Mod_Client[2].status,
                       ENO => #_w1);
   IF #_w1 AND #Mod_TCP_Setup.Mod_Client[2].error THEN
       #Mod_TCP_Setup.Mod_Client[2].statusSave := #Mod_TCP_Setup.Mod_Client[2].status;
   END_IF;
END_REGION

REGION Network 7: Read Master-2 Holding Register Value
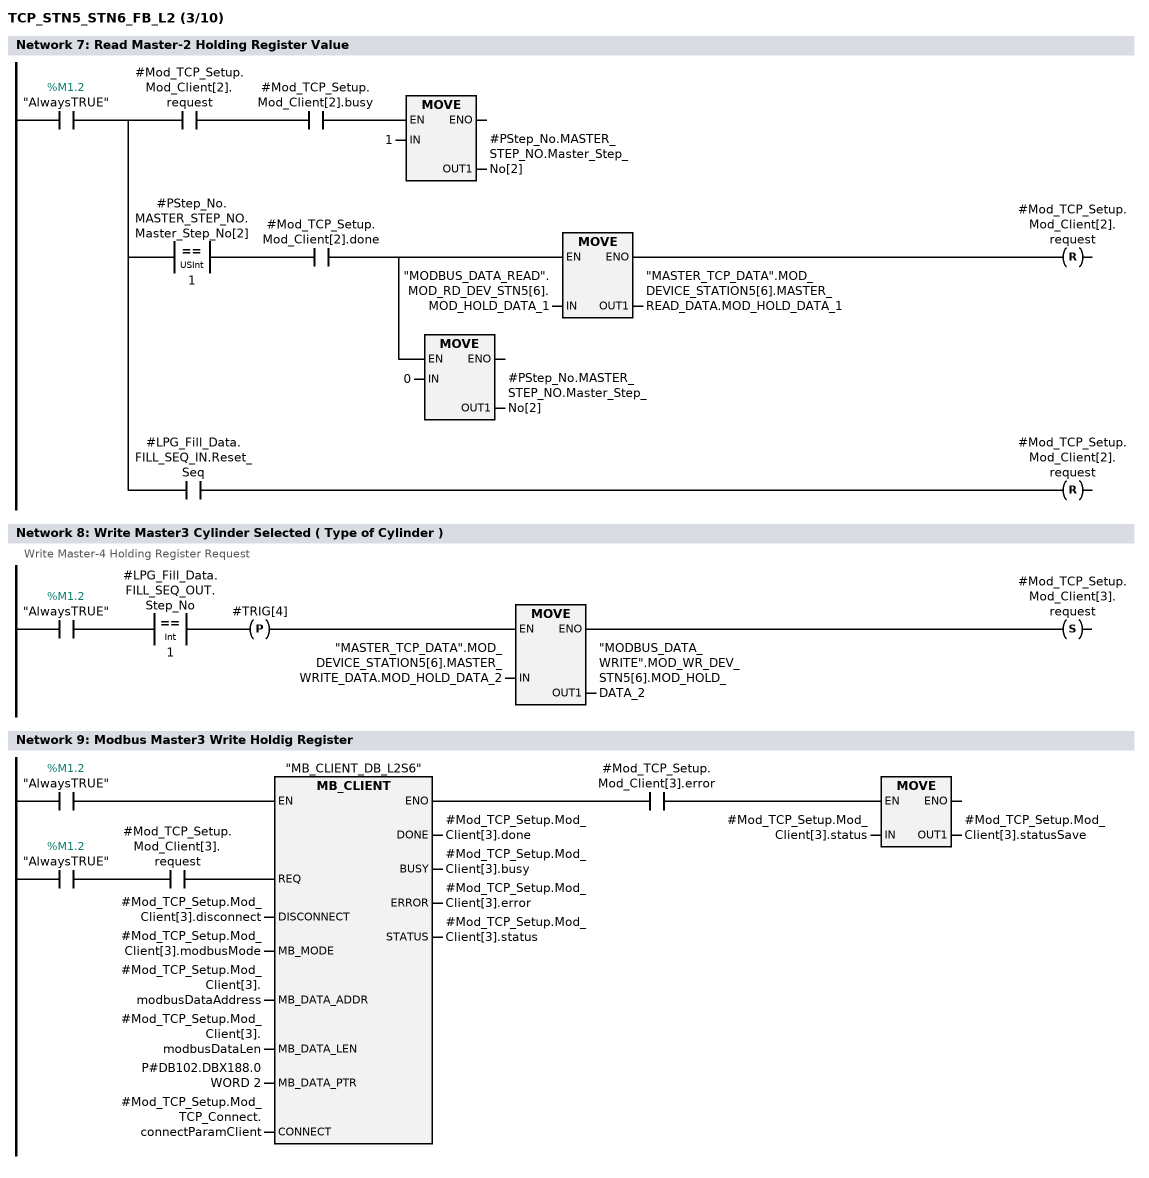
   RUNG wire#powerrail
      Contact( "AlwaysTRUE" )
      wire#w1
      Contact( #Mod_TCP_Setup.Mod_Client[2].request )
      Contact( #Mod_TCP_Setup.Mod_Client[2].busy )
      Move(in := 1, out1 => #PStep_No.MASTER_STEP_NO.Master_Step_No[2])
   END_RUNG
   RUNG wire#w1
      { S7_Templates := "SrcType := USInt" } EQ_Contact(in1 := #PStep_No.MASTER_STEP_NO.Master_Step_No[2], in2 := 1)
      Contact( #Mod_TCP_Setup.Mod_Client[2].done )
      wire#w2
      Move(in := "MODBUS_DATA_READ".MOD_RD_DEV_STN5[6].MOD_HOLD_DATA_1, out1 => "MASTER_TCP_DATA".MOD_DEVICE_STATION5[6].MASTER_READ_DATA.MOD_HOLD_DATA_1)
      R_Coil( #Mod_TCP_Setup.Mod_Client[2].request )
   END_RUNG
   RUNG wire#w2
      Move(in := 0, out1 => #PStep_No.MASTER_STEP_NO.Master_Step_No[2])
   END_RUNG
   RUNG wire#w1
      Contact( #LPG_Fill_Data.FILL_SEQ_IN.Reset_Seq )
      R_Coil( #Mod_TCP_Setup.Mod_Client[2].request )
   END_RUNG
   // the same network as SCL:
   IF "AlwaysTRUE" AND #Mod_TCP_Setup.Mod_Client[2].request AND #Mod_TCP_Setup.Mod_Client[2].busy THEN
       #PStep_No.MASTER_STEP_NO.Master_Step_No[2] := 1;
   END_IF;
   IF "AlwaysTRUE" AND (#PStep_No.MASTER_STEP_NO.Master_Step_No[2] = 1) AND #Mod_TCP_Setup.Mod_Client[2].done THEN
       "MASTER_TCP_DATA".MOD_DEVICE_STATION5[6].MASTER_READ_DATA.MOD_HOLD_DATA_1 := "MODBUS_DATA_READ".MOD_RD_DEV_STN5[6].MOD_HOLD_DATA_1;
   END_IF;
   #_w1 := "AlwaysTRUE" AND (#PStep_No.MASTER_STEP_NO.Master_Step_No[2] = 1) AND #Mod_TCP_Setup.Mod_Client[2].done;
   IF #_w1 THEN
       #Mod_TCP_Setup.Mod_Client[2].request := FALSE;
       #PStep_No.MASTER_STEP_NO.Master_Step_No[2] := 0;
   END_IF;
   IF "AlwaysTRUE" AND #LPG_Fill_Data.FILL_SEQ_IN.Reset_Seq THEN
       #Mod_TCP_Setup.Mod_Client[2].request := FALSE;
   END_IF;
END_REGION

REGION Network 8: Write Master3 Cylinder Selected ( Type of Cylinder )
   // Write Master-4 Holding Register Request
   RUNG wire#powerrail
      Contact( "AlwaysTRUE" )
      { S7_Templates := "SrcType := Int" } EQ_Contact(in1 := #LPG_Fill_Data.FILL_SEQ_OUT.Step_No, in2 := 1)
      P_Trig( #TRIG[4] )
      Move(in := "MASTER_TCP_DATA".MOD_DEVICE_STATION5[6].MASTER_WRITE_DATA.MOD_HOLD_DATA_2, out1 => "MODBUS_DATA_WRITE".MOD_WR_DEV_STN5[6].MOD_HOLD_DATA_2)
      S_Coil( #Mod_TCP_Setup.Mod_Client[3].request )
   END_RUNG
   // the same network as SCL:
   #_w1 := "AlwaysTRUE" AND (#LPG_Fill_Data.FILL_SEQ_OUT.Step_No = 1);
   #_w2 := #_w1 AND NOT #TRIG[4];   // rising edge
   #TRIG[4] := #_w1;
   IF #_w2 THEN
       "MODBUS_DATA_WRITE".MOD_WR_DEV_STN5[6].MOD_HOLD_DATA_2 := "MASTER_TCP_DATA".MOD_DEVICE_STATION5[6].MASTER_WRITE_DATA.MOD_HOLD_DATA_2;
       #Mod_TCP_Setup.Mod_Client[3].request := TRUE;
   END_IF;
END_REGION

REGION Network 9: Modbus Master3 Write Holdig Register
   RUNG wire#powerrail
      Contact( "AlwaysTRUE" )
      "MB_CLIENT_DB_L2S6".MB_CLIENT(REQ := wire#w1, DISCONNECT := #Mod_TCP_Setup.Mod_Client[3].disconnect, MB_MODE := #Mod_TCP_Setup.Mod_Client[3].modbusMode, MB_DATA_ADDR := #Mod_TCP_Setup.Mod_Client[3].modbusDataAddress, MB_DATA_LEN := #Mod_TCP_Setup.Mod_Client[3].modbusDataLen, MB_DATA_PTR := P#DB102.DBX188.0 WORD 2, CONNECT := #Mod_TCP_Setup.Mod_TCP_Connect.connectParamClient, DONE => #Mod_TCP_Setup.Mod_Client[3].done, BUSY => #Mod_TCP_Setup.Mod_Client[3].busy, ERROR => #Mod_TCP_Setup.Mod_Client[3].error, STATUS => #Mod_TCP_Setup.Mod_Client[3].status)
      Contact( #Mod_TCP_Setup.Mod_Client[3].error )
      Move(in := #Mod_TCP_Setup.Mod_Client[3].status, out1 => #Mod_TCP_Setup.Mod_Client[3].statusSave)
   END_RUNG
   RUNG wire#powerrail
      Contact( "AlwaysTRUE" )
      Contact( #Mod_TCP_Setup.Mod_Client[3].request )
   END_RUNG wire#w1
   // the same network as SCL:
   "MB_CLIENT_DB_L2S6"(EN := "AlwaysTRUE",   // MB_CLIENT
                       REQ := "AlwaysTRUE" AND #Mod_TCP_Setup.Mod_Client[3].request,
                       DISCONNECT := #Mod_TCP_Setup.Mod_Client[3].disconnect,
                       MB_MODE := #Mod_TCP_Setup.Mod_Client[3].modbusMode,
                       MB_DATA_ADDR := #Mod_TCP_Setup.Mod_Client[3].modbusDataAddress,
                       MB_DATA_LEN := #Mod_TCP_Setup.Mod_Client[3].modbusDataLen,
                       MB_DATA_PTR := P#DB102.DBX188.0 WORD 2,
                       CONNECT := #Mod_TCP_Setup.Mod_TCP_Connect.connectParamClient,
                       DONE => #Mod_TCP_Setup.Mod_Client[3].done,
                       BUSY => #Mod_TCP_Setup.Mod_Client[3].busy,
                       ERROR => #Mod_TCP_Setup.Mod_Client[3].error,
                       STATUS => #Mod_TCP_Setup.Mod_Client[3].status,
                       ENO => #_w1);
   IF #_w1 AND #Mod_TCP_Setup.Mod_Client[3].error THEN
       #Mod_TCP_Setup.Mod_Client[3].statusSave := #Mod_TCP_Setup.Mod_Client[3].status;
   END_IF;
END_REGION

REGION Network 10: Write Master-3 Holding Register Done
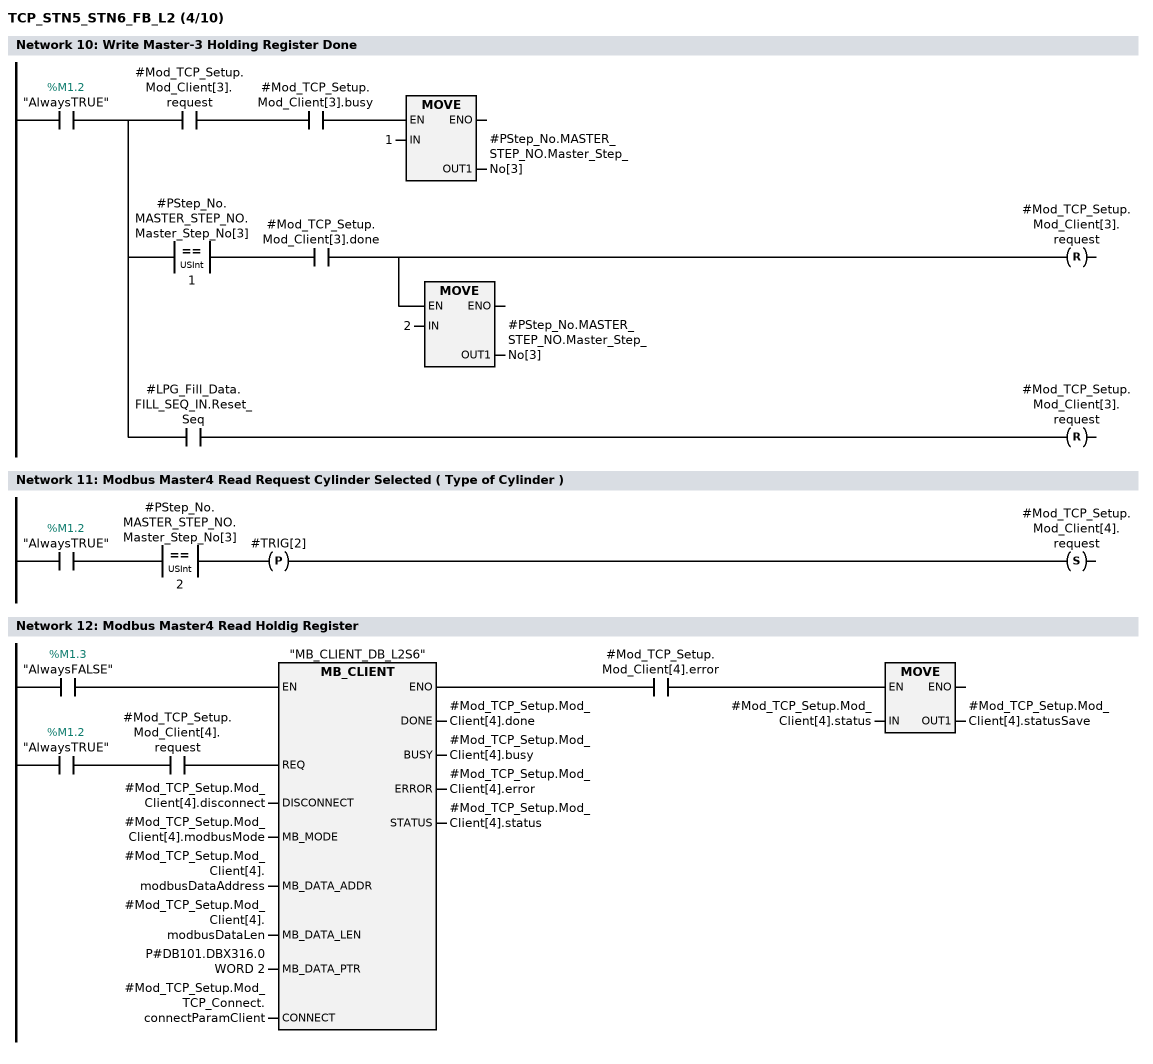
   RUNG wire#powerrail
      Contact( "AlwaysTRUE" )
      wire#w1
      Contact( #Mod_TCP_Setup.Mod_Client[3].request )
      Contact( #Mod_TCP_Setup.Mod_Client[3].busy )
      Move(in := 1, out1 => #PStep_No.MASTER_STEP_NO.Master_Step_No[3])
   END_RUNG
   RUNG wire#w1
      { S7_Templates := "SrcType := USInt" } EQ_Contact(in1 := #PStep_No.MASTER_STEP_NO.Master_Step_No[3], in2 := 1)
      Contact( #Mod_TCP_Setup.Mod_Client[3].done )
      wire#w2
      R_Coil( #Mod_TCP_Setup.Mod_Client[3].request )
   END_RUNG
   RUNG wire#w2
      Move(in := 2, out1 => #PStep_No.MASTER_STEP_NO.Master_Step_No[3])
   END_RUNG
   RUNG wire#w1
      Contact( #LPG_Fill_Data.FILL_SEQ_IN.Reset_Seq )
      R_Coil( #Mod_TCP_Setup.Mod_Client[3].request )
   END_RUNG
   // the same network as SCL:
   IF "AlwaysTRUE" AND #Mod_TCP_Setup.Mod_Client[3].request AND #Mod_TCP_Setup.Mod_Client[3].busy THEN
       #PStep_No.MASTER_STEP_NO.Master_Step_No[3] := 1;
   END_IF;
   #_w1 := "AlwaysTRUE" AND (#PStep_No.MASTER_STEP_NO.Master_Step_No[3] = 1) AND #Mod_TCP_Setup.Mod_Client[3].done;
   IF #_w1 THEN
       #Mod_TCP_Setup.Mod_Client[3].request := FALSE;
       #PStep_No.MASTER_STEP_NO.Master_Step_No[3] := 2;
   END_IF;
   IF "AlwaysTRUE" AND #LPG_Fill_Data.FILL_SEQ_IN.Reset_Seq THEN
       #Mod_TCP_Setup.Mod_Client[3].request := FALSE;
   END_IF;
END_REGION

REGION Network 11: Modbus Master4 Read Request Cylinder Selected ( Type of Cylinder )
   RUNG wire#powerrail
      Contact( "AlwaysTRUE" )
      { S7_Templates := "SrcType := USInt" } EQ_Contact(in1 := #PStep_No.MASTER_STEP_NO.Master_Step_No[3], in2 := 2)
      P_Trig( #TRIG[2] )
      S_Coil( #Mod_TCP_Setup.Mod_Client[4].request )
   END_RUNG
   // the same network as SCL:
   #_w1 := "AlwaysTRUE" AND (#PStep_No.MASTER_STEP_NO.Master_Step_No[3] = 2);
   #_w2 := #_w1 AND NOT #TRIG[2];   // rising edge
   #TRIG[2] := #_w1;
   IF #_w2 THEN #Mod_TCP_Setup.Mod_Client[4].request := TRUE; END_IF;
END_REGION

REGION Network 12: Modbus Master4 Read Holdig Register
   RUNG wire#powerrail
      Contact( "AlwaysFALSE" )
      "MB_CLIENT_DB_L2S6".MB_CLIENT(REQ := wire#w1, DISCONNECT := #Mod_TCP_Setup.Mod_Client[4].disconnect, MB_MODE := #Mod_TCP_Setup.Mod_Client[4].modbusMode, MB_DATA_ADDR := #Mod_TCP_Setup.Mod_Client[4].modbusDataAddress, MB_DATA_LEN := #Mod_TCP_Setup.Mod_Client[4].modbusDataLen, MB_DATA_PTR := P#DB101.DBX316.0 WORD 2, CONNECT := #Mod_TCP_Setup.Mod_TCP_Connect.connectParamClient, DONE => #Mod_TCP_Setup.Mod_Client[4].done, BUSY => #Mod_TCP_Setup.Mod_Client[4].busy, ERROR => #Mod_TCP_Setup.Mod_Client[4].error, STATUS => #Mod_TCP_Setup.Mod_Client[4].status)
      Contact( #Mod_TCP_Setup.Mod_Client[4].error )
      Move(in := #Mod_TCP_Setup.Mod_Client[4].status, out1 => #Mod_TCP_Setup.Mod_Client[4].statusSave)
   END_RUNG
   RUNG wire#powerrail
      Contact( "AlwaysTRUE" )
      Contact( #Mod_TCP_Setup.Mod_Client[4].request )
   END_RUNG wire#w1
   // the same network as SCL:
   "MB_CLIENT_DB_L2S6"(EN := "AlwaysFALSE",   // MB_CLIENT
                       REQ := "AlwaysTRUE" AND #Mod_TCP_Setup.Mod_Client[4].request,
                       DISCONNECT := #Mod_TCP_Setup.Mod_Client[4].disconnect,
                       MB_MODE := #Mod_TCP_Setup.Mod_Client[4].modbusMode,
                       MB_DATA_ADDR := #Mod_TCP_Setup.Mod_Client[4].modbusDataAddress,
                       MB_DATA_LEN := #Mod_TCP_Setup.Mod_Client[4].modbusDataLen,
                       MB_DATA_PTR := P#DB101.DBX316.0 WORD 2,
                       CONNECT := #Mod_TCP_Setup.Mod_TCP_Connect.connectParamClient,
                       DONE => #Mod_TCP_Setup.Mod_Client[4].done,
                       BUSY => #Mod_TCP_Setup.Mod_Client[4].busy,
                       ERROR => #Mod_TCP_Setup.Mod_Client[4].error,
                       STATUS => #Mod_TCP_Setup.Mod_Client[4].status,
                       ENO => #_w1);
   IF #_w1 AND #Mod_TCP_Setup.Mod_Client[4].error THEN
       #Mod_TCP_Setup.Mod_Client[4].statusSave := #Mod_TCP_Setup.Mod_Client[4].status;
   END_IF;
END_REGION

REGION Network 13: Read Master-4 Holding Register Value
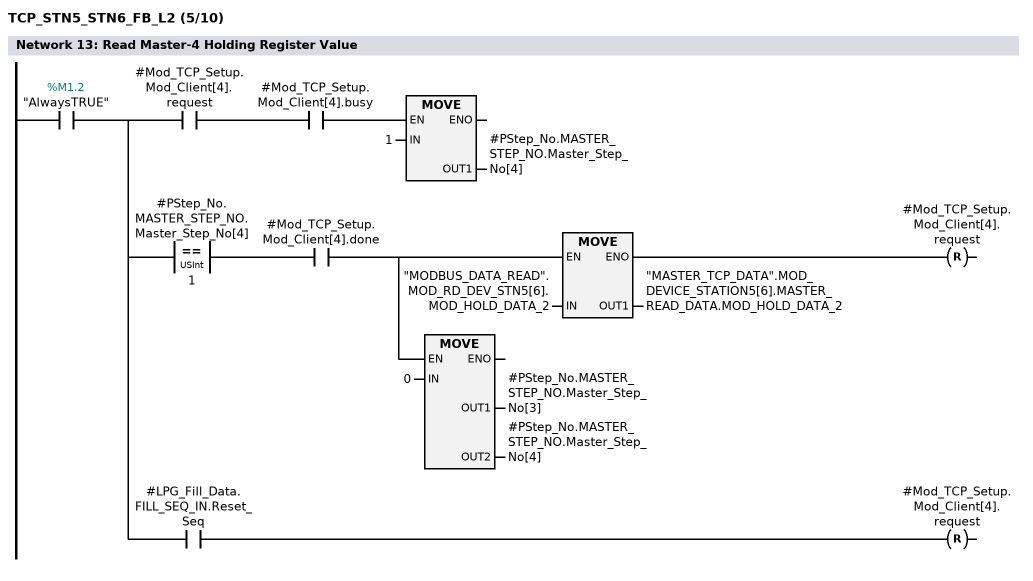
   RUNG wire#powerrail
      Contact( "AlwaysTRUE" )
      wire#w1
      Contact( #Mod_TCP_Setup.Mod_Client[4].request )
      Contact( #Mod_TCP_Setup.Mod_Client[4].busy )
      Move(in := 1, out1 => #PStep_No.MASTER_STEP_NO.Master_Step_No[4])
   END_RUNG
   RUNG wire#w1
      { S7_Templates := "SrcType := USInt" } EQ_Contact(in1 := #PStep_No.MASTER_STEP_NO.Master_Step_No[4], in2 := 1)
      Contact( #Mod_TCP_Setup.Mod_Client[4].done )
      wire#w2
      Move(in := "MODBUS_DATA_READ".MOD_RD_DEV_STN5[6].MOD_HOLD_DATA_2, out1 => "MASTER_TCP_DATA".MOD_DEVICE_STATION5[6].MASTER_READ_DATA.MOD_HOLD_DATA_2)
      R_Coil( #Mod_TCP_Setup.Mod_Client[4].request )
   END_RUNG
   RUNG wire#w2
      Move(in := 0, out1 => #PStep_No.MASTER_STEP_NO.Master_Step_No[3], out2 => #PStep_No.MASTER_STEP_NO.Master_Step_No[4])
   END_RUNG
   RUNG wire#w1
      Contact( #LPG_Fill_Data.FILL_SEQ_IN.Reset_Seq )
      R_Coil( #Mod_TCP_Setup.Mod_Client[4].request )
   END_RUNG
   // the same network as SCL:
   IF "AlwaysTRUE" AND #Mod_TCP_Setup.Mod_Client[4].request AND #Mod_TCP_Setup.Mod_Client[4].busy THEN
       #PStep_No.MASTER_STEP_NO.Master_Step_No[4] := 1;
   END_IF;
   IF "AlwaysTRUE" AND (#PStep_No.MASTER_STEP_NO.Master_Step_No[4] = 1) AND #Mod_TCP_Setup.Mod_Client[4].done THEN
       "MASTER_TCP_DATA".MOD_DEVICE_STATION5[6].MASTER_READ_DATA.MOD_HOLD_DATA_2 := "MODBUS_DATA_READ".MOD_RD_DEV_STN5[6].MOD_HOLD_DATA_2;
   END_IF;
   #_w1 := "AlwaysTRUE" AND (#PStep_No.MASTER_STEP_NO.Master_Step_No[4] = 1) AND #Mod_TCP_Setup.Mod_Client[4].done;
   IF #_w1 THEN
       #Mod_TCP_Setup.Mod_Client[4].request := FALSE;
       #PStep_No.MASTER_STEP_NO.Master_Step_No[3] := 0;
       #PStep_No.MASTER_STEP_NO.Master_Step_No[4] := 0;
   END_IF;
   IF "AlwaysTRUE" AND #LPG_Fill_Data.FILL_SEQ_IN.Reset_Seq THEN
       #Mod_TCP_Setup.Mod_Client[4].request := FALSE;
   END_IF;
END_REGION

REGION Network 14: Modbus Master5 Read Request(Coil Status)
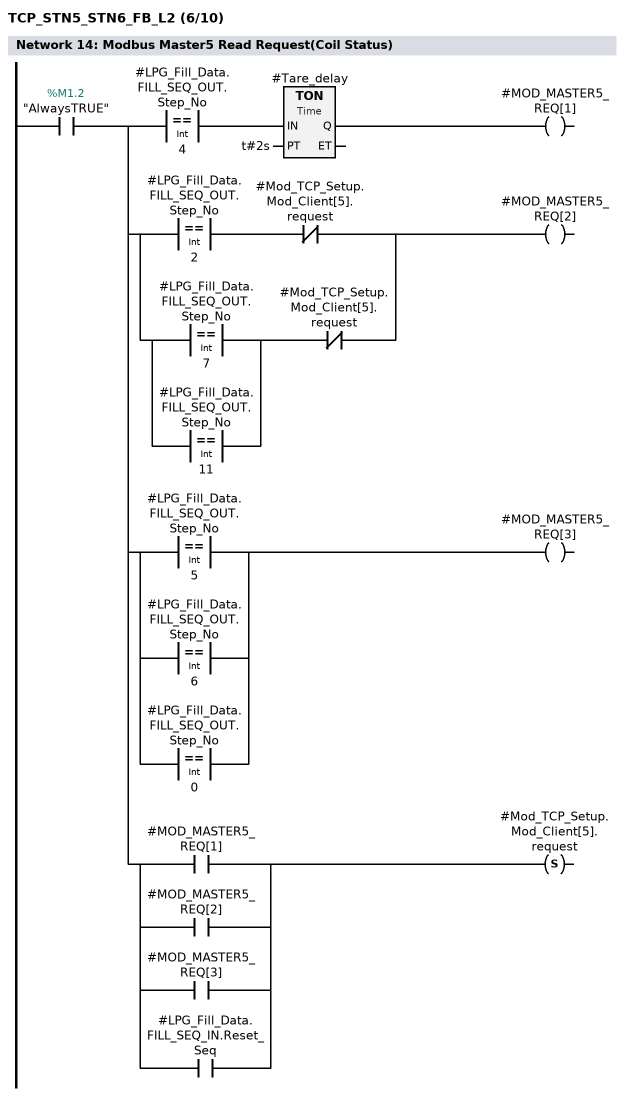
   RUNG wire#powerrail
      Contact( "AlwaysTRUE" )
      wire#w1
      { S7_Templates := "SrcType := Int" } EQ_Contact(in1 := #LPG_Fill_Data.FILL_SEQ_OUT.Step_No, in2 := 4)
      { S7_Templates := "time_type := Time" } #Tare_delay.TON(pt := t#2s, et =>)
      Coil( #MOD_MASTER5_REQ[1] )
   END_RUNG
   RUNG wire#w1
      { S7_Templates := "SrcType := Int" } EQ_Contact(in1 := #LPG_Fill_Data.FILL_SEQ_OUT.Step_No, in2 := 2)
      I_Contact( #Mod_TCP_Setup.Mod_Client[5].request )
      wire#w2
      Coil( #MOD_MASTER5_REQ[2] )
   END_RUNG
   RUNG wire#w1
      { S7_Templates := "SrcType := Int" } EQ_Contact(in1 := #LPG_Fill_Data.FILL_SEQ_OUT.Step_No, in2 := 7)
      wire#w3
      I_Contact( #Mod_TCP_Setup.Mod_Client[5].request )
   END_RUNG wire#w2
   RUNG wire#w1
      { S7_Templates := "SrcType := Int" } EQ_Contact(in1 := #LPG_Fill_Data.FILL_SEQ_OUT.Step_No, in2 := 11)
   END_RUNG wire#w3
   RUNG wire#w1
      { S7_Templates := "SrcType := Int" } EQ_Contact(in1 := #LPG_Fill_Data.FILL_SEQ_OUT.Step_No, in2 := 5)
      wire#w4
      Coil( #MOD_MASTER5_REQ[3] )
   END_RUNG
   RUNG wire#w1
      { S7_Templates := "SrcType := Int" } EQ_Contact(in1 := #LPG_Fill_Data.FILL_SEQ_OUT.Step_No, in2 := 6)
   END_RUNG wire#w4
   RUNG wire#w1
      { S7_Templates := "SrcType := Int" } EQ_Contact(in1 := #LPG_Fill_Data.FILL_SEQ_OUT.Step_No, in2 := 0)
   END_RUNG wire#w4
   RUNG wire#w1
      Contact( #MOD_MASTER5_REQ[1] )
      wire#w5
      S_Coil( #Mod_TCP_Setup.Mod_Client[5].request )
   END_RUNG
   RUNG wire#w1
      Contact( #MOD_MASTER5_REQ[2] )
   END_RUNG wire#w5
   RUNG wire#w1
      Contact( #MOD_MASTER5_REQ[3] )
   END_RUNG wire#w5
   RUNG wire#w1
      Contact( #LPG_Fill_Data.FILL_SEQ_IN.Reset_Seq )
   END_RUNG wire#w5
   // the same network as SCL:
   #Tare_delay(IN := "AlwaysTRUE" AND (#LPG_Fill_Data.FILL_SEQ_OUT.Step_No = 4), PT := t#2s);   // TON
   #MOD_MASTER5_REQ[1] := #Tare_delay.Q;
   #MOD_MASTER5_REQ[2] := "AlwaysTRUE" AND (((#LPG_Fill_Data.FILL_SEQ_OUT.Step_No = 2) AND NOT #Mod_TCP_Setup.Mod_Client[5].request) OR (((#LPG_Fill_Data.FILL_SEQ_OUT.Step_No = 7) OR (#LPG_Fill_Data.FILL_SEQ_OUT.Step_No = 11)) AND NOT #Mod_TCP_Setup.Mod_Client[5].request));
   #MOD_MASTER5_REQ[3] := "AlwaysTRUE" AND ((#LPG_Fill_Data.FILL_SEQ_OUT.Step_No = 5) OR (#LPG_Fill_Data.FILL_SEQ_OUT.Step_No = 6) OR (#LPG_Fill_Data.FILL_SEQ_OUT.Step_No = 0));
   IF "AlwaysTRUE" AND (#MOD_MASTER5_REQ[1] OR #MOD_MASTER5_REQ[2] OR #MOD_MASTER5_REQ[3] OR #LPG_Fill_Data.FILL_SEQ_IN.Reset_Seq) THEN
       #Mod_TCP_Setup.Mod_Client[5].request := TRUE;
   END_IF;
END_REGION

REGION Network 15: Modbus Master5 Read Coil Status
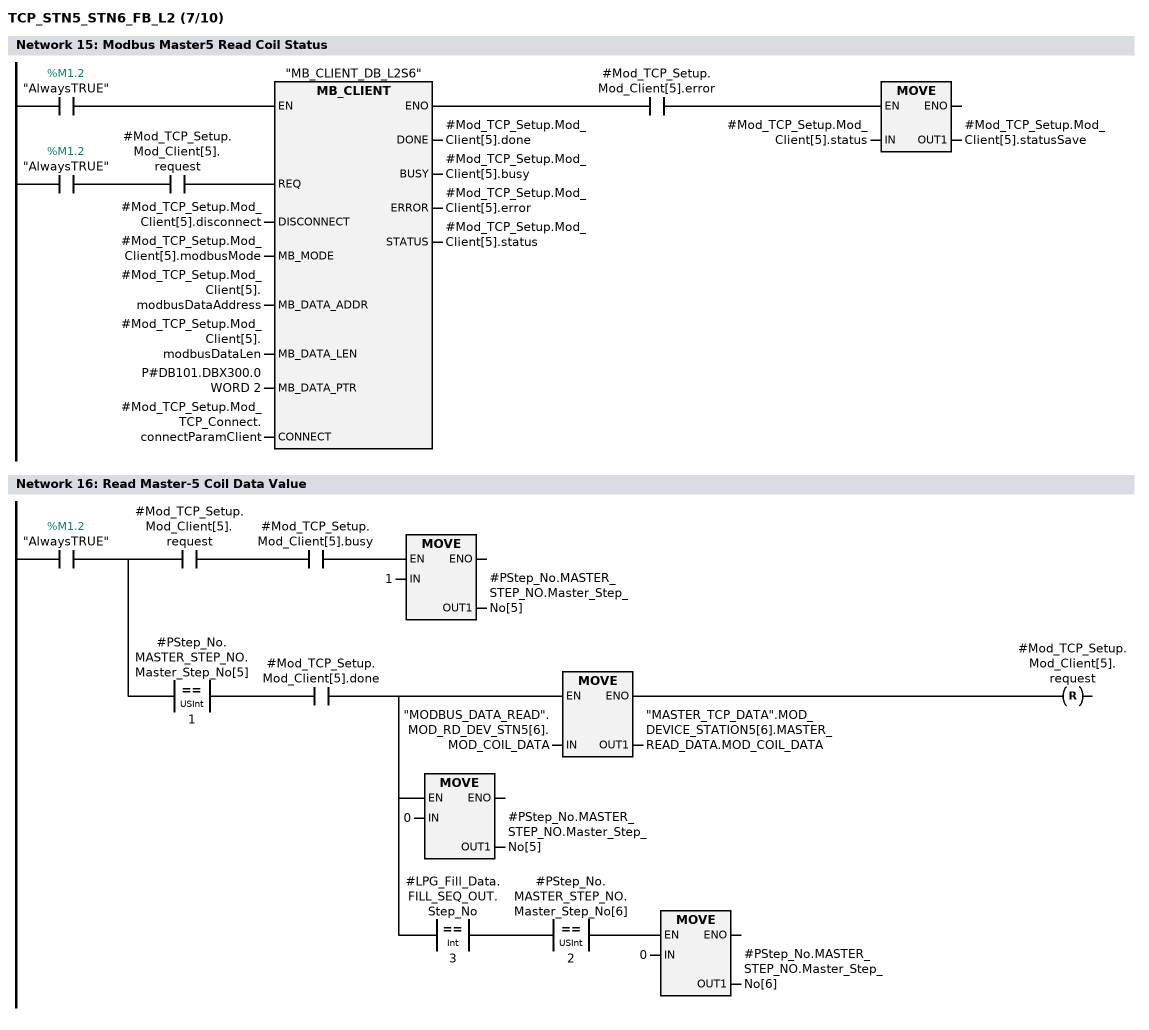
   RUNG wire#powerrail
      Contact( "AlwaysTRUE" )
      "MB_CLIENT_DB_L2S6".MB_CLIENT(REQ := wire#w1, DISCONNECT := #Mod_TCP_Setup.Mod_Client[5].disconnect, MB_MODE := #Mod_TCP_Setup.Mod_Client[5].modbusMode, MB_DATA_ADDR := #Mod_TCP_Setup.Mod_Client[5].modbusDataAddress, MB_DATA_LEN := #Mod_TCP_Setup.Mod_Client[5].modbusDataLen, MB_DATA_PTR := P#DB101.DBX300.0 WORD 2, CONNECT := #Mod_TCP_Setup.Mod_TCP_Connect.connectParamClient, DONE => #Mod_TCP_Setup.Mod_Client[5].done, BUSY => #Mod_TCP_Setup.Mod_Client[5].busy, ERROR => #Mod_TCP_Setup.Mod_Client[5].error, STATUS => #Mod_TCP_Setup.Mod_Client[5].status)
      Contact( #Mod_TCP_Setup.Mod_Client[5].error )
      Move(in := #Mod_TCP_Setup.Mod_Client[5].status, out1 => #Mod_TCP_Setup.Mod_Client[5].statusSave)
   END_RUNG
   RUNG wire#powerrail
      Contact( "AlwaysTRUE" )
      Contact( #Mod_TCP_Setup.Mod_Client[5].request )
   END_RUNG wire#w1
   // the same network as SCL:
   "MB_CLIENT_DB_L2S6"(EN := "AlwaysTRUE",   // MB_CLIENT
                       REQ := "AlwaysTRUE" AND #Mod_TCP_Setup.Mod_Client[5].request,
                       DISCONNECT := #Mod_TCP_Setup.Mod_Client[5].disconnect,
                       MB_MODE := #Mod_TCP_Setup.Mod_Client[5].modbusMode,
                       MB_DATA_ADDR := #Mod_TCP_Setup.Mod_Client[5].modbusDataAddress,
                       MB_DATA_LEN := #Mod_TCP_Setup.Mod_Client[5].modbusDataLen,
                       MB_DATA_PTR := P#DB101.DBX300.0 WORD 2,
                       CONNECT := #Mod_TCP_Setup.Mod_TCP_Connect.connectParamClient,
                       DONE => #Mod_TCP_Setup.Mod_Client[5].done,
                       BUSY => #Mod_TCP_Setup.Mod_Client[5].busy,
                       ERROR => #Mod_TCP_Setup.Mod_Client[5].error,
                       STATUS => #Mod_TCP_Setup.Mod_Client[5].status,
                       ENO => #_w1);
   IF #_w1 AND #Mod_TCP_Setup.Mod_Client[5].error THEN
       #Mod_TCP_Setup.Mod_Client[5].statusSave := #Mod_TCP_Setup.Mod_Client[5].status;
   END_IF;
END_REGION

REGION Network 16: Read Master-5 Coil Data Value
   RUNG wire#powerrail
      Contact( "AlwaysTRUE" )
      wire#w1
      Contact( #Mod_TCP_Setup.Mod_Client[5].request )
      Contact( #Mod_TCP_Setup.Mod_Client[5].busy )
      Move(in := 1, out1 => #PStep_No.MASTER_STEP_NO.Master_Step_No[5])
   END_RUNG
   RUNG wire#w1
      { S7_Templates := "SrcType := USInt" } EQ_Contact(in1 := #PStep_No.MASTER_STEP_NO.Master_Step_No[5], in2 := 1)
      Contact( #Mod_TCP_Setup.Mod_Client[5].done )
      wire#w2
      Move(in := "MODBUS_DATA_READ".MOD_RD_DEV_STN5[6].MOD_COIL_DATA, out1 => "MASTER_TCP_DATA".MOD_DEVICE_STATION5[6].MASTER_READ_DATA.MOD_COIL_DATA)
      R_Coil( #Mod_TCP_Setup.Mod_Client[5].request )
   END_RUNG
   RUNG wire#w2
      Move(in := 0, out1 => #PStep_No.MASTER_STEP_NO.Master_Step_No[5])
   END_RUNG
   RUNG wire#w2
      { S7_Templates := "SrcType := Int" } EQ_Contact(in1 := #LPG_Fill_Data.FILL_SEQ_OUT.Step_No, in2 := 3)
      { S7_Templates := "SrcType := USInt" } EQ_Contact(in1 := #PStep_No.MASTER_STEP_NO.Master_Step_No[6], in2 := 2)
      Move(in := 0, out1 => #PStep_No.MASTER_STEP_NO.Master_Step_No[6])
   END_RUNG
   // the same network as SCL:
   IF "AlwaysTRUE" AND #Mod_TCP_Setup.Mod_Client[5].request AND #Mod_TCP_Setup.Mod_Client[5].busy THEN
       #PStep_No.MASTER_STEP_NO.Master_Step_No[5] := 1;
   END_IF;
   #_w1 := "AlwaysTRUE" AND (#PStep_No.MASTER_STEP_NO.Master_Step_No[5] = 1) AND #Mod_TCP_Setup.Mod_Client[5].done;
   IF #_w1 THEN
       "MASTER_TCP_DATA".MOD_DEVICE_STATION5[6].MASTER_READ_DATA.MOD_COIL_DATA := "MODBUS_DATA_READ".MOD_RD_DEV_STN5[6].MOD_COIL_DATA;
       #Mod_TCP_Setup.Mod_Client[5].request := FALSE;
       #PStep_No.MASTER_STEP_NO.Master_Step_No[5] := 0;
   END_IF;
   IF #_w1 AND (#LPG_Fill_Data.FILL_SEQ_OUT.Step_No = 3) AND (#PStep_No.MASTER_STEP_NO.Master_Step_No[6] = 2) THEN
       #PStep_No.MASTER_STEP_NO.Master_Step_No[6] := 0;
   END_IF;
END_REGION

REGION Network 17: Write Coil Data
   // if multiple bit write not working
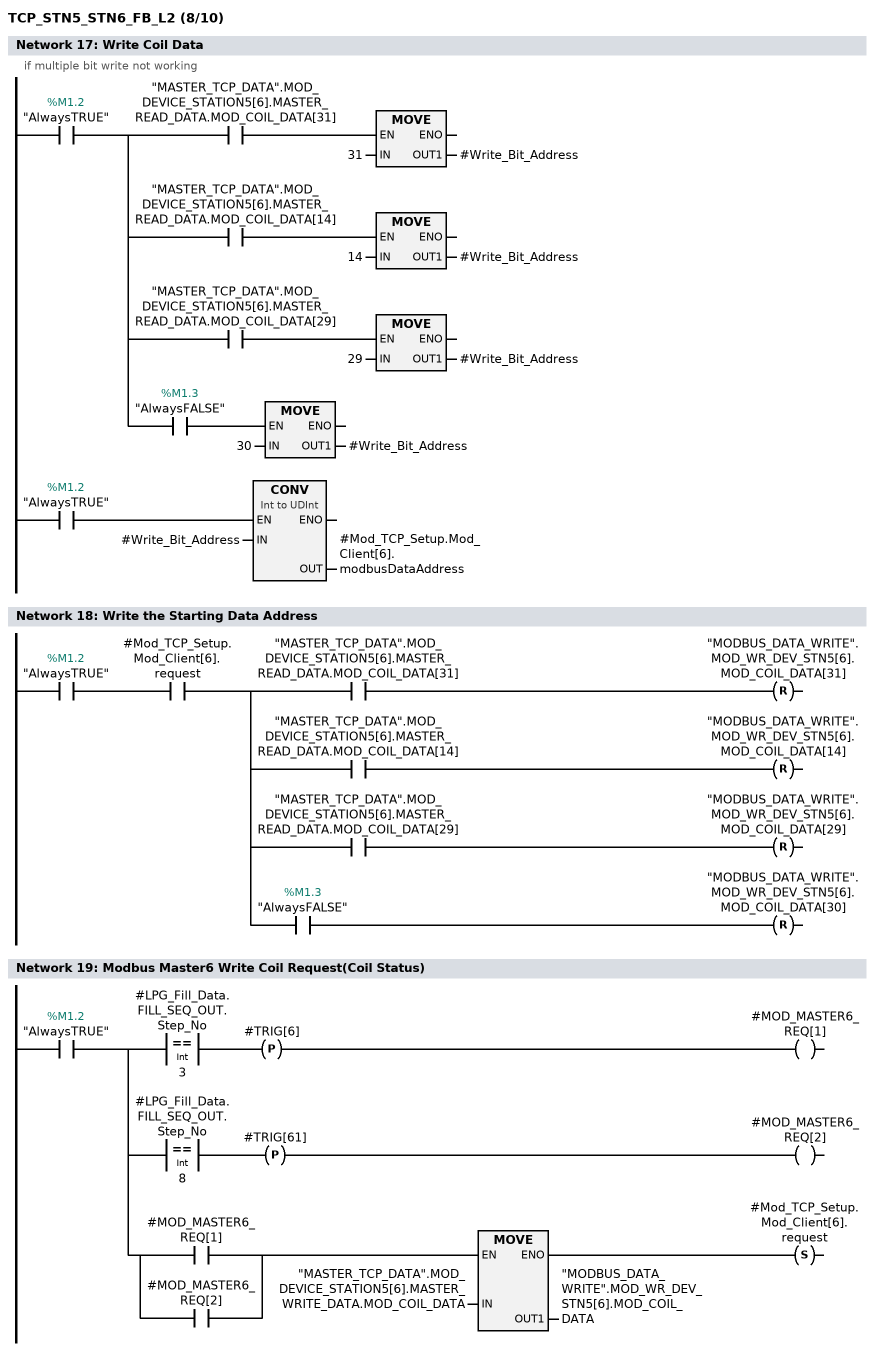
   RUNG wire#powerrail
      Contact( "AlwaysTRUE" )
      wire#w1
      Contact( "MASTER_TCP_DATA".MOD_DEVICE_STATION5[6].MASTER_READ_DATA.MOD_COIL_DATA[31] )
      Move(in := 31, out1 => #Write_Bit_Address)
   END_RUNG
   RUNG wire#w1
      Contact( "MASTER_TCP_DATA".MOD_DEVICE_STATION5[6].MASTER_READ_DATA.MOD_COIL_DATA[14] )
      Move(in := 14, out1 => #Write_Bit_Address)
   END_RUNG
   RUNG wire#w1
      Contact( "MASTER_TCP_DATA".MOD_DEVICE_STATION5[6].MASTER_READ_DATA.MOD_COIL_DATA[29] )
      Move(in := 29, out1 => #Write_Bit_Address)
   END_RUNG
   RUNG wire#w1
      Contact( "AlwaysFALSE" )
      Move(in := 30, out1 => #Write_Bit_Address)
   END_RUNG
   RUNG wire#powerrail
      Contact( "AlwaysTRUE" )
      { S7_Templates := "[SrcType := Int, DestType := UDInt]" } Convert(in := #Write_Bit_Address, out => #Mod_TCP_Setup.Mod_Client[6].modbusDataAddress)
   END_RUNG
   // the same network as SCL:
   IF "AlwaysTRUE" AND "MASTER_TCP_DATA".MOD_DEVICE_STATION5[6].MASTER_READ_DATA.MOD_COIL_DATA[31] THEN
       #Write_Bit_Address := 31;
   END_IF;
   IF "AlwaysTRUE" AND "MASTER_TCP_DATA".MOD_DEVICE_STATION5[6].MASTER_READ_DATA.MOD_COIL_DATA[14] THEN
       #Write_Bit_Address := 14;
   END_IF;
   IF "AlwaysTRUE" AND "MASTER_TCP_DATA".MOD_DEVICE_STATION5[6].MASTER_READ_DATA.MOD_COIL_DATA[29] THEN
       #Write_Bit_Address := 29;
   END_IF;
   IF "AlwaysTRUE" AND "AlwaysFALSE" THEN #Write_Bit_Address := 30; END_IF;
   IF "AlwaysTRUE" THEN
       #Mod_TCP_Setup.Mod_Client[6].modbusDataAddress := INT_TO_UDINT(#Write_Bit_Address);
   END_IF;
END_REGION

REGION Network 18: Write the Starting Data Address
   RUNG wire#powerrail
      Contact( "AlwaysTRUE" )
      Contact( #Mod_TCP_Setup.Mod_Client[6].request )
      wire#w1
      Contact( "MASTER_TCP_DATA".MOD_DEVICE_STATION5[6].MASTER_READ_DATA.MOD_COIL_DATA[31] )
      R_Coil( "MODBUS_DATA_WRITE".MOD_WR_DEV_STN5[6].MOD_COIL_DATA[31] )
   END_RUNG
   RUNG wire#w1
      Contact( "MASTER_TCP_DATA".MOD_DEVICE_STATION5[6].MASTER_READ_DATA.MOD_COIL_DATA[14] )
      R_Coil( "MODBUS_DATA_WRITE".MOD_WR_DEV_STN5[6].MOD_COIL_DATA[14] )
   END_RUNG
   RUNG wire#w1
      Contact( "MASTER_TCP_DATA".MOD_DEVICE_STATION5[6].MASTER_READ_DATA.MOD_COIL_DATA[29] )
      R_Coil( "MODBUS_DATA_WRITE".MOD_WR_DEV_STN5[6].MOD_COIL_DATA[29] )
   END_RUNG
   RUNG wire#w1
      Contact( "AlwaysFALSE" )
      R_Coil( "MODBUS_DATA_WRITE".MOD_WR_DEV_STN5[6].MOD_COIL_DATA[30] )
   END_RUNG
   // the same network as SCL:
   #_w1 := "AlwaysTRUE" AND #Mod_TCP_Setup.Mod_Client[6].request;
   IF #_w1 AND "MASTER_TCP_DATA".MOD_DEVICE_STATION5[6].MASTER_READ_DATA.MOD_COIL_DATA[31] THEN
       "MODBUS_DATA_WRITE".MOD_WR_DEV_STN5[6].MOD_COIL_DATA[31] := FALSE;
   END_IF;
   IF #_w1 AND "MASTER_TCP_DATA".MOD_DEVICE_STATION5[6].MASTER_READ_DATA.MOD_COIL_DATA[14] THEN
       "MODBUS_DATA_WRITE".MOD_WR_DEV_STN5[6].MOD_COIL_DATA[14] := FALSE;
   END_IF;
   IF #_w1 AND "MASTER_TCP_DATA".MOD_DEVICE_STATION5[6].MASTER_READ_DATA.MOD_COIL_DATA[29] THEN
       "MODBUS_DATA_WRITE".MOD_WR_DEV_STN5[6].MOD_COIL_DATA[29] := FALSE;
   END_IF;
   IF #_w1 AND "AlwaysFALSE" THEN "MODBUS_DATA_WRITE".MOD_WR_DEV_STN5[6].MOD_COIL_DATA[30] := FALSE; END_IF;
END_REGION

REGION Network 19: Modbus Master6 Write Coil Request(Coil Status)
   RUNG wire#powerrail
      Contact( "AlwaysTRUE" )
      wire#w1
      { S7_Templates := "SrcType := Int" } EQ_Contact(in1 := #LPG_Fill_Data.FILL_SEQ_OUT.Step_No, in2 := 3)
      P_Trig( #TRIG[6] )
      Coil( #MOD_MASTER6_REQ[1] )
   END_RUNG
   RUNG wire#w1
      { S7_Templates := "SrcType := Int" } EQ_Contact(in1 := #LPG_Fill_Data.FILL_SEQ_OUT.Step_No, in2 := 8)
      P_Trig( #TRIG[61] )
      Coil( #MOD_MASTER6_REQ[2] )
   END_RUNG
   RUNG wire#w1
      Contact( #MOD_MASTER6_REQ[1] )
      wire#w2
      Move(in := "MASTER_TCP_DATA".MOD_DEVICE_STATION5[6].MASTER_WRITE_DATA.MOD_COIL_DATA, out1 => "MODBUS_DATA_WRITE".MOD_WR_DEV_STN5[6].MOD_COIL_DATA)
      S_Coil( #Mod_TCP_Setup.Mod_Client[6].request )
   END_RUNG
   RUNG wire#w1
      Contact( #MOD_MASTER6_REQ[2] )
   END_RUNG wire#w2
   // the same network as SCL:
   #_w1 := "AlwaysTRUE" AND (#LPG_Fill_Data.FILL_SEQ_OUT.Step_No = 3);
   #_w2 := #_w1 AND NOT #TRIG[6];   // rising edge
   #TRIG[6] := #_w1;
   #MOD_MASTER6_REQ[1] := #_w2;
   #_w3 := "AlwaysTRUE" AND (#LPG_Fill_Data.FILL_SEQ_OUT.Step_No = 8);
   #_w4 := #_w3 AND NOT #TRIG[61];   // rising edge
   #TRIG[61] := #_w3;
   #MOD_MASTER6_REQ[2] := #_w4;
   IF "AlwaysTRUE" AND (#MOD_MASTER6_REQ[1] OR #MOD_MASTER6_REQ[2]) THEN
       "MODBUS_DATA_WRITE".MOD_WR_DEV_STN5[6].MOD_COIL_DATA := "MASTER_TCP_DATA".MOD_DEVICE_STATION5[6].MASTER_WRITE_DATA.MOD_COIL_DATA;
       #Mod_TCP_Setup.Mod_Client[6].request := TRUE;
   END_IF;
END_REGION

REGION Network 20: Modbus Master6 Write Coil Status
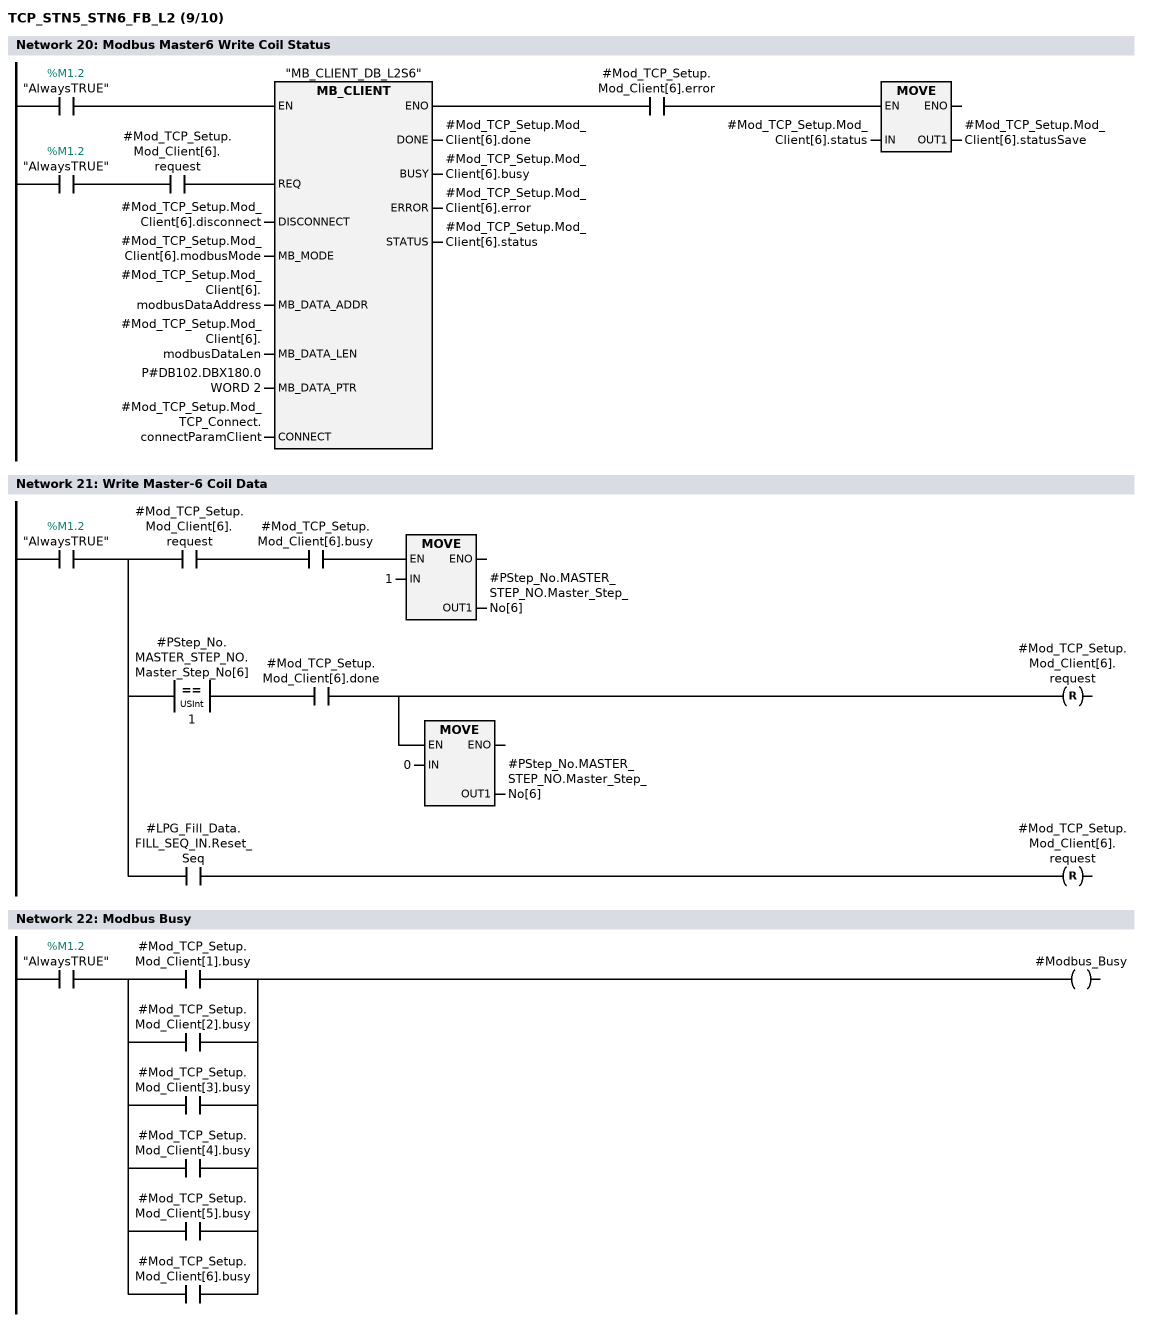
   RUNG wire#powerrail
      Contact( "AlwaysTRUE" )
      "MB_CLIENT_DB_L2S6".MB_CLIENT(REQ := wire#w1, DISCONNECT := #Mod_TCP_Setup.Mod_Client[6].disconnect, MB_MODE := #Mod_TCP_Setup.Mod_Client[6].modbusMode, MB_DATA_ADDR := #Mod_TCP_Setup.Mod_Client[6].modbusDataAddress, MB_DATA_LEN := #Mod_TCP_Setup.Mod_Client[6].modbusDataLen, MB_DATA_PTR := P#DB102.DBX180.0 WORD 2, CONNECT := #Mod_TCP_Setup.Mod_TCP_Connect.connectParamClient, DONE => #Mod_TCP_Setup.Mod_Client[6].done, BUSY => #Mod_TCP_Setup.Mod_Client[6].busy, ERROR => #Mod_TCP_Setup.Mod_Client[6].error, STATUS => #Mod_TCP_Setup.Mod_Client[6].status)
      Contact( #Mod_TCP_Setup.Mod_Client[6].error )
      Move(in := #Mod_TCP_Setup.Mod_Client[6].status, out1 => #Mod_TCP_Setup.Mod_Client[6].statusSave)
   END_RUNG
   RUNG wire#powerrail
      Contact( "AlwaysTRUE" )
      Contact( #Mod_TCP_Setup.Mod_Client[6].request )
   END_RUNG wire#w1
   // the same network as SCL:
   "MB_CLIENT_DB_L2S6"(EN := "AlwaysTRUE",   // MB_CLIENT
                       REQ := "AlwaysTRUE" AND #Mod_TCP_Setup.Mod_Client[6].request,
                       DISCONNECT := #Mod_TCP_Setup.Mod_Client[6].disconnect,
                       MB_MODE := #Mod_TCP_Setup.Mod_Client[6].modbusMode,
                       MB_DATA_ADDR := #Mod_TCP_Setup.Mod_Client[6].modbusDataAddress,
                       MB_DATA_LEN := #Mod_TCP_Setup.Mod_Client[6].modbusDataLen,
                       MB_DATA_PTR := P#DB102.DBX180.0 WORD 2,
                       CONNECT := #Mod_TCP_Setup.Mod_TCP_Connect.connectParamClient,
                       DONE => #Mod_TCP_Setup.Mod_Client[6].done,
                       BUSY => #Mod_TCP_Setup.Mod_Client[6].busy,
                       ERROR => #Mod_TCP_Setup.Mod_Client[6].error,
                       STATUS => #Mod_TCP_Setup.Mod_Client[6].status,
                       ENO => #_w1);
   IF #_w1 AND #Mod_TCP_Setup.Mod_Client[6].error THEN
       #Mod_TCP_Setup.Mod_Client[6].statusSave := #Mod_TCP_Setup.Mod_Client[6].status;
   END_IF;
END_REGION

REGION Network 21: Write Master-6 Coil Data
   RUNG wire#powerrail
      Contact( "AlwaysTRUE" )
      wire#w1
      Contact( #Mod_TCP_Setup.Mod_Client[6].request )
      Contact( #Mod_TCP_Setup.Mod_Client[6].busy )
      Move(in := 1, out1 => #PStep_No.MASTER_STEP_NO.Master_Step_No[6])
   END_RUNG
   RUNG wire#w1
      { S7_Templates := "SrcType := USInt" } EQ_Contact(in1 := #PStep_No.MASTER_STEP_NO.Master_Step_No[6], in2 := 1)
      Contact( #Mod_TCP_Setup.Mod_Client[6].done )
      wire#w2
      R_Coil( #Mod_TCP_Setup.Mod_Client[6].request )
   END_RUNG
   RUNG wire#w2
      Move(in := 0, out1 => #PStep_No.MASTER_STEP_NO.Master_Step_No[6])
   END_RUNG
   RUNG wire#w1
      Contact( #LPG_Fill_Data.FILL_SEQ_IN.Reset_Seq )
      R_Coil( #Mod_TCP_Setup.Mod_Client[6].request )
   END_RUNG
   // the same network as SCL:
   IF "AlwaysTRUE" AND #Mod_TCP_Setup.Mod_Client[6].request AND #Mod_TCP_Setup.Mod_Client[6].busy THEN
       #PStep_No.MASTER_STEP_NO.Master_Step_No[6] := 1;
   END_IF;
   #_w1 := "AlwaysTRUE" AND (#PStep_No.MASTER_STEP_NO.Master_Step_No[6] = 1) AND #Mod_TCP_Setup.Mod_Client[6].done;
   IF #_w1 THEN
       #Mod_TCP_Setup.Mod_Client[6].request := FALSE;
       #PStep_No.MASTER_STEP_NO.Master_Step_No[6] := 0;
   END_IF;
   IF "AlwaysTRUE" AND #LPG_Fill_Data.FILL_SEQ_IN.Reset_Seq THEN
       #Mod_TCP_Setup.Mod_Client[6].request := FALSE;
   END_IF;
END_REGION

REGION Network 22: Modbus Busy
   RUNG wire#powerrail
      Contact( "AlwaysTRUE" )
      wire#w1
      Contact( #Mod_TCP_Setup.Mod_Client[1].busy )
      wire#w2
      Coil( #Modbus_Busy )
   END_RUNG
   RUNG wire#w1
      Contact( #Mod_TCP_Setup.Mod_Client[2].busy )
   END_RUNG wire#w2
   RUNG wire#w1
      Contact( #Mod_TCP_Setup.Mod_Client[3].busy )
   END_RUNG wire#w2
   RUNG wire#w1
      Contact( #Mod_TCP_Setup.Mod_Client[4].busy )
   END_RUNG wire#w2
   RUNG wire#w1
      Contact( #Mod_TCP_Setup.Mod_Client[5].busy )
   END_RUNG wire#w2
   RUNG wire#w1
      Contact( #Mod_TCP_Setup.Mod_Client[6].busy )
   END_RUNG wire#w2
   // the same network as SCL:
   #Modbus_Busy := "AlwaysTRUE" AND (#Mod_TCP_Setup.Mod_Client[1].busy OR #Mod_TCP_Setup.Mod_Client[2].busy OR #Mod_TCP_Setup.Mod_Client[3].busy OR #Mod_TCP_Setup.Mod_Client[4].busy OR #Mod_TCP_Setup.Mod_Client[5].busy OR #Mod_TCP_Setup.Mod_Client[6].busy);
END_REGION

REGION Network 23
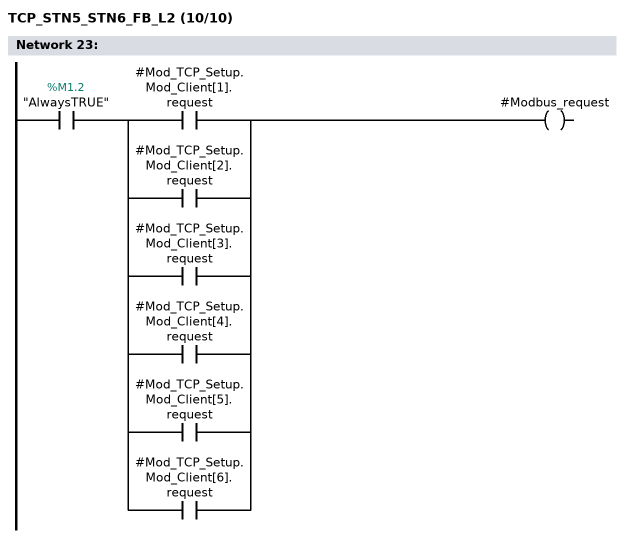
   RUNG wire#powerrail
      Contact( "AlwaysTRUE" )
      wire#w1
      Contact( #Mod_TCP_Setup.Mod_Client[1].request )
      wire#w2
      Coil( #Modbus_request )
   END_RUNG
   RUNG wire#w1
      Contact( #Mod_TCP_Setup.Mod_Client[2].request )
   END_RUNG wire#w2
   RUNG wire#w1
      Contact( #Mod_TCP_Setup.Mod_Client[3].request )
   END_RUNG wire#w2
   RUNG wire#w1
      Contact( #Mod_TCP_Setup.Mod_Client[4].request )
   END_RUNG wire#w2
   RUNG wire#w1
      Contact( #Mod_TCP_Setup.Mod_Client[5].request )
   END_RUNG wire#w2
   RUNG wire#w1
      Contact( #Mod_TCP_Setup.Mod_Client[6].request )
   END_RUNG wire#w2
   // the same network as SCL:
   #Modbus_request := "AlwaysTRUE" AND (#Mod_TCP_Setup.Mod_Client[1].request OR #Mod_TCP_Setup.Mod_Client[2].request OR #Mod_TCP_Setup.Mod_Client[3].request OR #Mod_TCP_Setup.Mod_Client[4].request OR #Mod_TCP_Setup.Mod_Client[5].request OR #Mod_TCP_Setup.Mod_Client[6].request);
END_REGION
END_FUNCTION_BLOCK

FUNCTION "Common_Logoc" : Void   // FC1, LAD
{ S7_Optimized_Access := 'TRUE' }
VERSION : 0.1
// stored: AutoNumber true, IsIECCheckEnabled false, SetENOAutomatically false, UDAEnableTagReadback false
BEGIN

REGION Network 1: Empty Network
   // Ohm Namashivaya
END_REGION

REGION Network 2: Total Enabled Stations
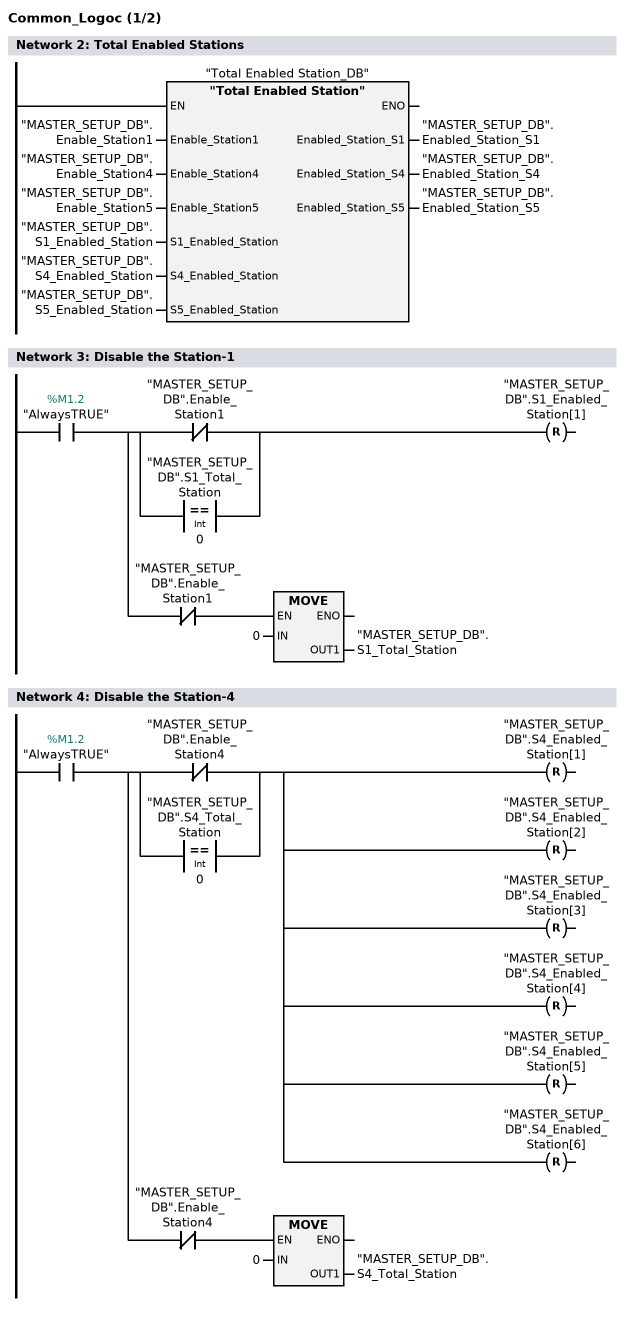
   RUNG wire#powerrail
      "Total Enabled Station_DB"(Enable_Station1 := "MASTER_SETUP_DB".Enable_Station1, Enable_Station4 := "MASTER_SETUP_DB".Enable_Station4, Enable_Station5 := "MASTER_SETUP_DB".Enable_Station5, S1_Enabled_Station := "MASTER_SETUP_DB".S1_Enabled_Station, S4_Enabled_Station := "MASTER_SETUP_DB".S4_Enabled_Station, S5_Enabled_Station := "MASTER_SETUP_DB".S5_Enabled_Station, Enabled_Station_S1 => "MASTER_SETUP_DB".Enabled_Station_S1, Enabled_Station_S4 => "MASTER_SETUP_DB".Enabled_Station_S4, Enabled_Station_S5 => "MASTER_SETUP_DB".Enabled_Station_S5)
   END_RUNG
   // the same network as SCL:
   "Total Enabled Station_DB"(Enable_Station1 := "MASTER_SETUP_DB".Enable_Station1,   // "Total Enabled Station"
                           Enable_Station4 := "MASTER_SETUP_DB".Enable_Station4,
                           Enable_Station5 := "MASTER_SETUP_DB".Enable_Station5,
                           S1_Enabled_Station := "MASTER_SETUP_DB".S1_Enabled_Station,
                           S4_Enabled_Station := "MASTER_SETUP_DB".S4_Enabled_Station,
                           S5_Enabled_Station := "MASTER_SETUP_DB".S5_Enabled_Station,
                           Enabled_Station_S1 => "MASTER_SETUP_DB".Enabled_Station_S1,
                           Enabled_Station_S4 => "MASTER_SETUP_DB".Enabled_Station_S4,
                           Enabled_Station_S5 => "MASTER_SETUP_DB".Enabled_Station_S5);
END_REGION

REGION Network 3: Disable the Station-1
   RUNG wire#powerrail
      Contact( "AlwaysTRUE" )
      wire#w1
      I_Contact( "MASTER_SETUP_DB".Enable_Station1 )
      wire#w2
      R_Coil( "MASTER_SETUP_DB".S1_Enabled_Station[1] )
   END_RUNG
   RUNG wire#w1
      { S7_Templates := "SrcType := Int" } EQ_Contact(in1 := "MASTER_SETUP_DB".S1_Total_Station, in2 := 0)
   END_RUNG wire#w2
   RUNG wire#w1
      I_Contact( "MASTER_SETUP_DB".Enable_Station1 )
      Move(in := 0, out1 => "MASTER_SETUP_DB".S1_Total_Station)
   END_RUNG
   // the same network as SCL:
   IF "AlwaysTRUE" AND (NOT "MASTER_SETUP_DB".Enable_Station1 OR ("MASTER_SETUP_DB".S1_Total_Station = 0)) THEN
       "MASTER_SETUP_DB".S1_Enabled_Station[1] := FALSE;
   END_IF;
   IF "AlwaysTRUE" AND NOT "MASTER_SETUP_DB".Enable_Station1 THEN
       "MASTER_SETUP_DB".S1_Total_Station := 0;
   END_IF;
END_REGION

REGION Network 4: Disable the Station-4
   RUNG wire#powerrail
      Contact( "AlwaysTRUE" )
      wire#w1
      I_Contact( "MASTER_SETUP_DB".Enable_Station4 )
      wire#w2
      R_Coil( "MASTER_SETUP_DB".S4_Enabled_Station[1] )
   END_RUNG
   RUNG wire#w1
      { S7_Templates := "SrcType := Int" } EQ_Contact(in1 := "MASTER_SETUP_DB".S4_Total_Station, in2 := 0)
   END_RUNG wire#w2
   RUNG wire#w2
      R_Coil( "MASTER_SETUP_DB".S4_Enabled_Station[2] )
   END_RUNG
   RUNG wire#w2
      R_Coil( "MASTER_SETUP_DB".S4_Enabled_Station[3] )
   END_RUNG
   RUNG wire#w2
      R_Coil( "MASTER_SETUP_DB".S4_Enabled_Station[4] )
   END_RUNG
   RUNG wire#w2
      R_Coil( "MASTER_SETUP_DB".S4_Enabled_Station[5] )
   END_RUNG
   RUNG wire#w2
      R_Coil( "MASTER_SETUP_DB".S4_Enabled_Station[6] )
   END_RUNG
   RUNG wire#w1
      I_Contact( "MASTER_SETUP_DB".Enable_Station4 )
      Move(in := 0, out1 => "MASTER_SETUP_DB".S4_Total_Station)
   END_RUNG
   // the same network as SCL:
   IF "AlwaysTRUE" AND (NOT "MASTER_SETUP_DB".Enable_Station4 OR ("MASTER_SETUP_DB".S4_Total_Station = 0)) THEN
       "MASTER_SETUP_DB".S4_Enabled_Station[1] := FALSE;
       "MASTER_SETUP_DB".S4_Enabled_Station[2] := FALSE;
       "MASTER_SETUP_DB".S4_Enabled_Station[3] := FALSE;
       "MASTER_SETUP_DB".S4_Enabled_Station[4] := FALSE;
       "MASTER_SETUP_DB".S4_Enabled_Station[5] := FALSE;
       "MASTER_SETUP_DB".S4_Enabled_Station[6] := FALSE;
   END_IF;
   IF "AlwaysTRUE" AND NOT "MASTER_SETUP_DB".Enable_Station4 THEN
       "MASTER_SETUP_DB".S4_Total_Station := 0;
   END_IF;
END_REGION

REGION Network 5: Disable the Station-5
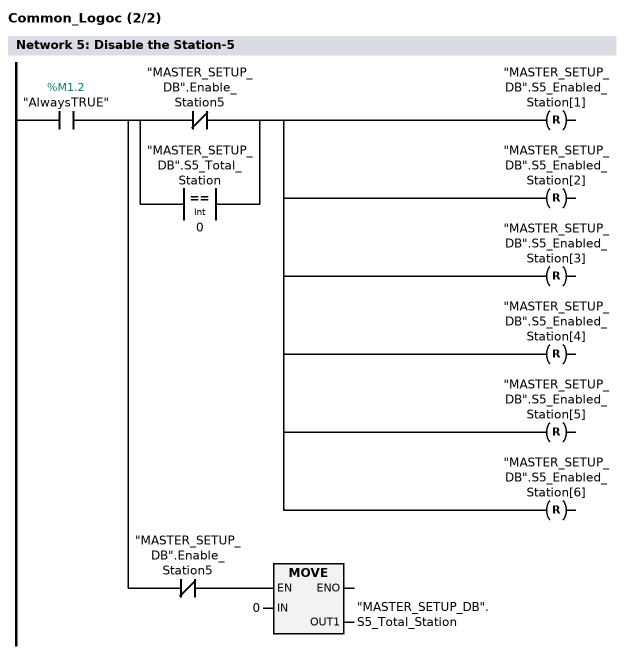
   RUNG wire#powerrail
      Contact( "AlwaysTRUE" )
      wire#w1
      I_Contact( "MASTER_SETUP_DB".Enable_Station5 )
      wire#w2
      R_Coil( "MASTER_SETUP_DB".S5_Enabled_Station[1] )
   END_RUNG
   RUNG wire#w1
      { S7_Templates := "SrcType := Int" } EQ_Contact(in1 := "MASTER_SETUP_DB".S5_Total_Station, in2 := 0)
   END_RUNG wire#w2
   RUNG wire#w2
      R_Coil( "MASTER_SETUP_DB".S5_Enabled_Station[2] )
   END_RUNG
   RUNG wire#w2
      R_Coil( "MASTER_SETUP_DB".S5_Enabled_Station[3] )
   END_RUNG
   RUNG wire#w2
      R_Coil( "MASTER_SETUP_DB".S5_Enabled_Station[4] )
   END_RUNG
   RUNG wire#w2
      R_Coil( "MASTER_SETUP_DB".S5_Enabled_Station[5] )
   END_RUNG
   RUNG wire#w2
      R_Coil( "MASTER_SETUP_DB".S5_Enabled_Station[6] )
   END_RUNG
   RUNG wire#w1
      I_Contact( "MASTER_SETUP_DB".Enable_Station5 )
      Move(in := 0, out1 => "MASTER_SETUP_DB".S5_Total_Station)
   END_RUNG
   // the same network as SCL:
   IF "AlwaysTRUE" AND (NOT "MASTER_SETUP_DB".Enable_Station5 OR ("MASTER_SETUP_DB".S5_Total_Station = 0)) THEN
       "MASTER_SETUP_DB".S5_Enabled_Station[1] := FALSE;
       "MASTER_SETUP_DB".S5_Enabled_Station[2] := FALSE;
       "MASTER_SETUP_DB".S5_Enabled_Station[3] := FALSE;
       "MASTER_SETUP_DB".S5_Enabled_Station[4] := FALSE;
       "MASTER_SETUP_DB".S5_Enabled_Station[5] := FALSE;
       "MASTER_SETUP_DB".S5_Enabled_Station[6] := FALSE;
   END_IF;
   IF "AlwaysTRUE" AND NOT "MASTER_SETUP_DB".Enable_Station5 THEN
       "MASTER_SETUP_DB".S5_Total_Station := 0;
   END_IF;
END_REGION
END_FUNCTION

FUNCTION_BLOCK "Total Enabled Station"   // FB9, LAD
{ S7_Optimized_Access := 'TRUE' }
VERSION : 0.1
// stored: AutoNumber true, IsIECCheckEnabled false, IsRetainMemResEnabled false, MemoryReserve 100, SetENOAutomatically false, UDAEnableTagReadback false
   VAR_INPUT
      Enable_Station1 : Bool;
      Enable_Station4 : Bool;
      Enable_Station5 : Bool;
      S1_Enabled_Station : Array[1..6] of Bool;
      S4_Enabled_Station : Array[1..6] of Bool;
      S5_Enabled_Station : Array[1..6] of Bool;
   END_VAR
   VAR_OUTPUT
      Enabled_Station_S1 : Int;
      Enabled_Station_S4 : Int;
      Enabled_Station_S5 : Int;
   END_VAR
   VAR
      Enabled_Station1 { S7_SetPoint := 'True'} : "Enabled_Station";
      Enabled_Station4 { S7_SetPoint := 'True'} : "Enabled_Station";
      Enabled_Station5 { S7_SetPoint := 'True'} : "Enabled_Station";
   END_VAR
BEGIN

REGION Network 2: s1
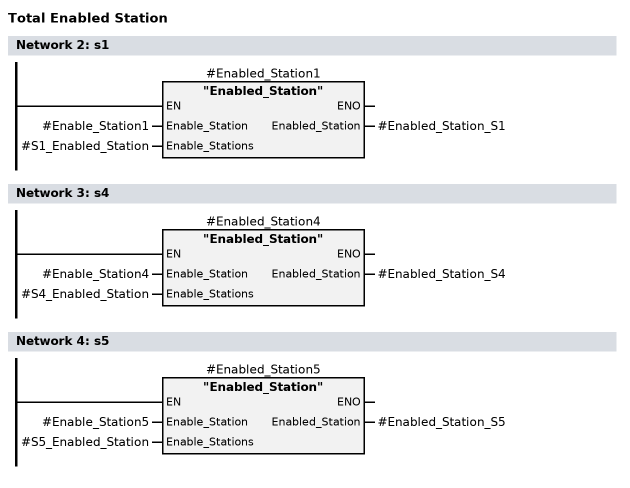
   RUNG wire#powerrail
      #Enabled_Station1(Enable_Station := #Enable_Station1, Enable_Stations := #S1_Enabled_Station, Enabled_Station => #Enabled_Station_S1)
   END_RUNG
   // the same network as SCL:
   #Enabled_Station1(Enable_Station := #Enable_Station1,   // "Enabled_Station"
                     Enable_Stations := #S1_Enabled_Station,
                     Enabled_Station => #Enabled_Station_S1);
END_REGION

REGION Network 3: s4
   RUNG wire#powerrail
      #Enabled_Station4(Enable_Station := #Enable_Station4, Enable_Stations := #S4_Enabled_Station, Enabled_Station => #Enabled_Station_S4)
   END_RUNG
   // the same network as SCL:
   #Enabled_Station4(Enable_Station := #Enable_Station4,   // "Enabled_Station"
                     Enable_Stations := #S4_Enabled_Station,
                     Enabled_Station => #Enabled_Station_S4);
END_REGION

REGION Network 4: s5
   RUNG wire#powerrail
      #Enabled_Station5(Enable_Station := #Enable_Station5, Enable_Stations := #S5_Enabled_Station, Enabled_Station => #Enabled_Station_S5)
   END_RUNG
   // the same network as SCL:
   #Enabled_Station5(Enable_Station := #Enable_Station5,   // "Enabled_Station"
                     Enable_Stations := #S5_Enabled_Station,
                     Enabled_Station => #Enabled_Station_S5);
END_REGION
END_FUNCTION_BLOCK

FUNCTION_BLOCK "Enabled_Station"   // FB2, LAD
{ S7_Optimized_Access := 'TRUE' }
VERSION : 0.1
// stored: AutoNumber true, IsIECCheckEnabled false, IsRetainMemResEnabled false, MemoryReserve 100, SetENOAutomatically false, UDAEnableTagReadback false
   VAR_INPUT
      Enable_Station : Bool;
      Enable_Stations : Array[1..6] of Bool;
   END_VAR
   VAR_OUTPUT
      Enabled_Station : Int;
   END_VAR
   VAR
      Station1 : Int;
      Station2 : Int;
      Station3 : Int;
      Station4 : Int;
      Station5 : Int;
      Station6 : Int;
   END_VAR
   VAR_TEMP   // added for the SCL form of the ladder/FBD networks
      _w1 : Bool;
   END_VAR
BEGIN

REGION Network 2: Station-1 Enabled
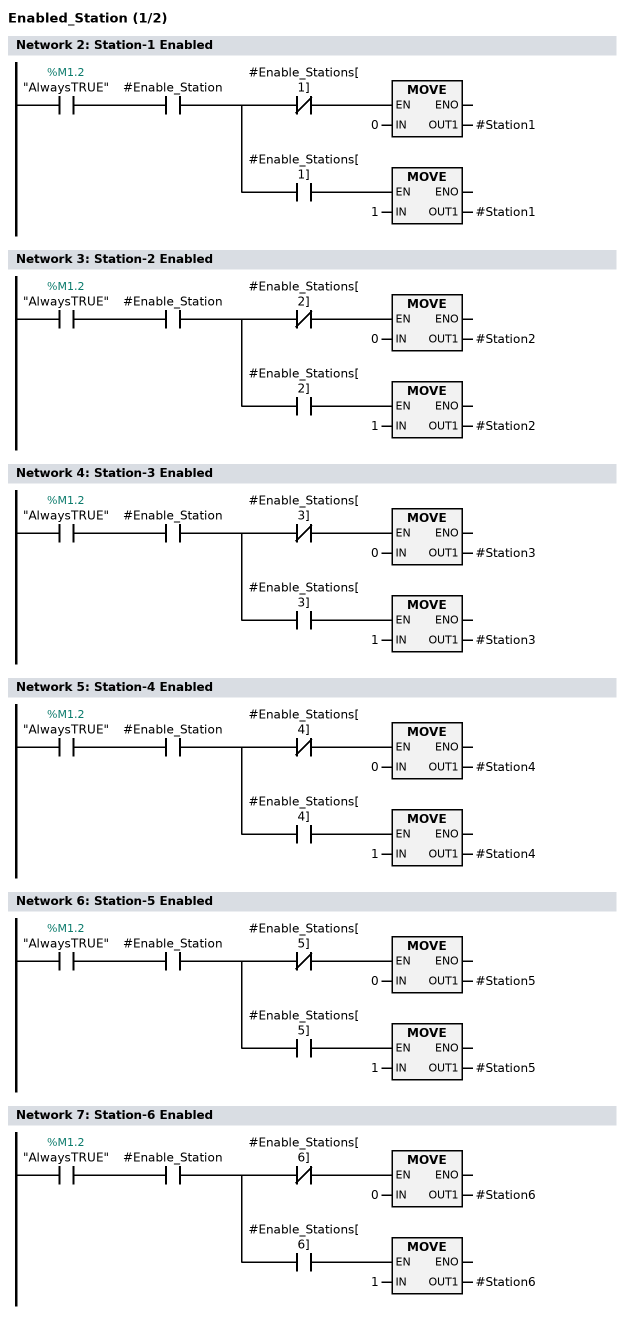
   RUNG wire#powerrail
      Contact( "AlwaysTRUE" )
      Contact( #Enable_Station )
      wire#w1
      I_Contact( #Enable_Stations[1] )
      Move(in := 0, out1 => #Station1)
   END_RUNG
   RUNG wire#w1
      Contact( #Enable_Stations[1] )
      Move(in := 1, out1 => #Station1)
   END_RUNG
   // the same network as SCL:
   #_w1 := "AlwaysTRUE" AND #Enable_Station;
   IF #_w1 AND NOT #Enable_Stations[1] THEN #Station1 := 0; END_IF;
   IF #_w1 AND #Enable_Stations[1] THEN #Station1 := 1; END_IF;
END_REGION

REGION Network 3: Station-2 Enabled
   RUNG wire#powerrail
      Contact( "AlwaysTRUE" )
      Contact( #Enable_Station )
      wire#w1
      I_Contact( #Enable_Stations[2] )
      Move(in := 0, out1 => #Station2)
   END_RUNG
   RUNG wire#w1
      Contact( #Enable_Stations[2] )
      Move(in := 1, out1 => #Station2)
   END_RUNG
   // the same network as SCL:
   #_w1 := "AlwaysTRUE" AND #Enable_Station;
   IF #_w1 AND NOT #Enable_Stations[2] THEN #Station2 := 0; END_IF;
   IF #_w1 AND #Enable_Stations[2] THEN #Station2 := 1; END_IF;
END_REGION

REGION Network 4: Station-3 Enabled
   RUNG wire#powerrail
      Contact( "AlwaysTRUE" )
      Contact( #Enable_Station )
      wire#w1
      I_Contact( #Enable_Stations[3] )
      Move(in := 0, out1 => #Station3)
   END_RUNG
   RUNG wire#w1
      Contact( #Enable_Stations[3] )
      Move(in := 1, out1 => #Station3)
   END_RUNG
   // the same network as SCL:
   #_w1 := "AlwaysTRUE" AND #Enable_Station;
   IF #_w1 AND NOT #Enable_Stations[3] THEN #Station3 := 0; END_IF;
   IF #_w1 AND #Enable_Stations[3] THEN #Station3 := 1; END_IF;
END_REGION

REGION Network 5: Station-4 Enabled
   RUNG wire#powerrail
      Contact( "AlwaysTRUE" )
      Contact( #Enable_Station )
      wire#w1
      I_Contact( #Enable_Stations[4] )
      Move(in := 0, out1 => #Station4)
   END_RUNG
   RUNG wire#w1
      Contact( #Enable_Stations[4] )
      Move(in := 1, out1 => #Station4)
   END_RUNG
   // the same network as SCL:
   #_w1 := "AlwaysTRUE" AND #Enable_Station;
   IF #_w1 AND NOT #Enable_Stations[4] THEN #Station4 := 0; END_IF;
   IF #_w1 AND #Enable_Stations[4] THEN #Station4 := 1; END_IF;
END_REGION

REGION Network 6: Station-5 Enabled
   RUNG wire#powerrail
      Contact( "AlwaysTRUE" )
      Contact( #Enable_Station )
      wire#w1
      I_Contact( #Enable_Stations[5] )
      Move(in := 0, out1 => #Station5)
   END_RUNG
   RUNG wire#w1
      Contact( #Enable_Stations[5] )
      Move(in := 1, out1 => #Station5)
   END_RUNG
   // the same network as SCL:
   #_w1 := "AlwaysTRUE" AND #Enable_Station;
   IF #_w1 AND NOT #Enable_Stations[5] THEN #Station5 := 0; END_IF;
   IF #_w1 AND #Enable_Stations[5] THEN #Station5 := 1; END_IF;
END_REGION

REGION Network 7: Station-6 Enabled
   RUNG wire#powerrail
      Contact( "AlwaysTRUE" )
      Contact( #Enable_Station )
      wire#w1
      I_Contact( #Enable_Stations[6] )
      Move(in := 0, out1 => #Station6)
   END_RUNG
   RUNG wire#w1
      Contact( #Enable_Stations[6] )
      Move(in := 1, out1 => #Station6)
   END_RUNG
   // the same network as SCL:
   #_w1 := "AlwaysTRUE" AND #Enable_Station;
   IF #_w1 AND NOT #Enable_Stations[6] THEN #Station6 := 0; END_IF;
   IF #_w1 AND #Enable_Stations[6] THEN #Station6 := 1; END_IF;
END_REGION

REGION Network 8
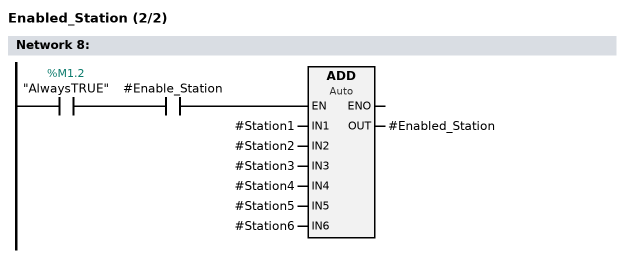
   RUNG wire#powerrail
      Contact( "AlwaysTRUE" )
      Contact( #Enable_Station )
      Add(in1 := #Station1, in2 := #Station2, in3 := #Station3, in4 := #Station4, in5 := #Station5, in6 := #Station6, out => #Enabled_Station)
   END_RUNG
   // the same network as SCL:
   IF "AlwaysTRUE" AND #Enable_Station THEN
       #Enabled_Station := #Station1 + #Station2 + #Station3 + #Station4 + #Station5 + #Station6;
   END_IF;
END_REGION
END_FUNCTION_BLOCK

FUNCTION_BLOCK "FILLING_STATION4_FB"   // FB500, LAD
{ S7_Optimized_Access := 'TRUE' }
VERSION : 0.1
// stored: AutoNumber false, IsIECCheckEnabled false, IsRetainMemResEnabled false, MemoryReserve 100, SetENOAutomatically false, UDAEnableTagReadback false
   VAR
      STATION4_S1 { S7_SetPoint := 'True'} : "LPG_FILLING_FB";
      STATION4_S2 { S7_SetPoint := 'True'} : "LPG_FILLING_FB";
      STATION4_S3 { S7_SetPoint := 'True'} : "LPG_FILLING_FB";
      STATION4_S4 { S7_SetPoint := 'True'} : "LPG_FILLING_FB";
      STATION4_S5 { S7_SetPoint := 'True'} : "LPG_FILLING_FB";
      STATION4_S6 { S7_SetPoint := 'True'} : "LPG_FILLING_FB";
      FILLING_STATION4 { S7_SetPoint := 'True'} : "FILLING_FB";
      FILL_SEQ_STARTED { S7_SetPoint := 'True'} : Array[1..6] of Bool;
      FILLING_DONE : Array[1..6] of Bool;
   END_VAR
   VAR_TEMP   // added for the SCL form of the ladder/FBD networks
      _w1 : Bool;
   END_VAR
BEGIN

REGION Network 2: Call Filling Station-4
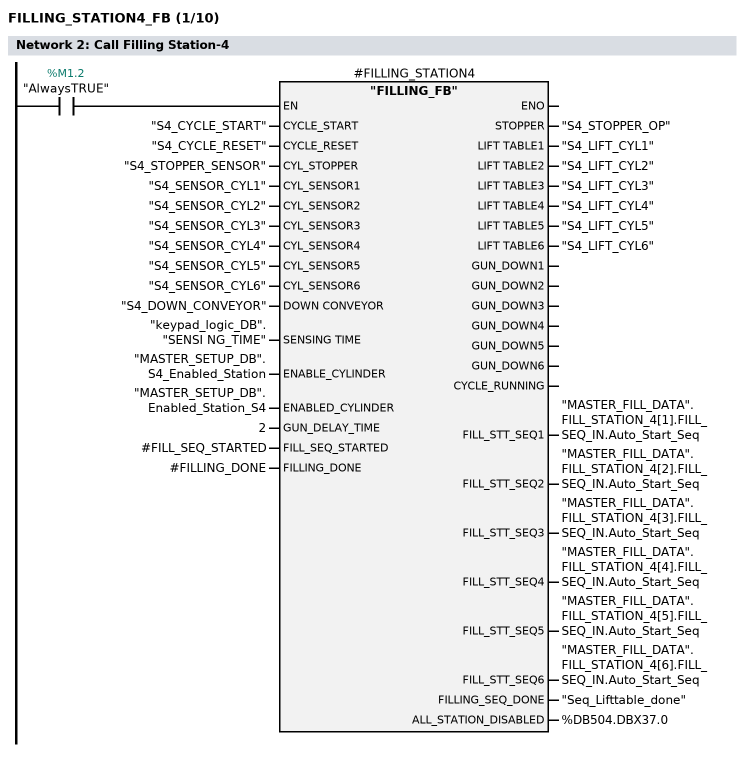
   RUNG wire#powerrail
      Contact( "AlwaysTRUE" )
      #FILLING_STATION4(CYCLE_START := "S4_CYCLE_START", CYCLE_RESET := "S4_CYCLE_RESET", CYL_STOPPER := "S4_STOPPER_SENSOR", CYL_SENSOR1 := "S4_SENSOR_CYL1", CYL_SENSOR2 := "S4_SENSOR_CYL2", CYL_SENSOR3 := "S4_SENSOR_CYL3", CYL_SENSOR4 := "S4_SENSOR_CYL4", CYL_SENSOR5 := "S4_SENSOR_CYL5", CYL_SENSOR6 := "S4_SENSOR_CYL6", "DOWN CONVEYOR" := "S4_DOWN_CONVEYOR", "SENSING TIME" := "keypad_logic_DB"."SENSI NG_TIME", ENABLE_CYLINDER := "MASTER_SETUP_DB".S4_Enabled_Station, ENABLED_CYLINDER := "MASTER_SETUP_DB".Enabled_Station_S4, GUN_DELAY_TIME := 2, FILL_SEQ_STARTED := #FILL_SEQ_STARTED, FILLING_DONE := #FILLING_DONE, STOPPER => "S4_STOPPER_OP", "LIFT TABLE1" => "S4_LIFT_CYL1", "LIFT TABLE2" => "S4_LIFT_CYL2", "LIFT TABLE3" => "S4_LIFT_CYL3", "LIFT TABLE4" => "S4_LIFT_CYL4", "LIFT TABLE5" => "S4_LIFT_CYL5", "LIFT TABLE6" => "S4_LIFT_CYL6", GUN_DOWN1 =>, GUN_DOWN2 =>, GUN_DOWN3 =>, GUN_DOWN4 =>, GUN_DOWN5 =>, GUN_DOWN6 =>, CYCLE_RUNNING =>, FILL_STT_SEQ1 => "MASTER_FILL_DATA".FILL_STATION_4[1].FILL_SEQ_IN.Auto_Start_Seq, FILL_STT_SEQ2 => "MASTER_FILL_DATA".FILL_STATION_4[2].FILL_SEQ_IN.Auto_Start_Seq, FILL_STT_SEQ3 => "MASTER_FILL_DATA".FILL_STATION_4[3].FILL_SEQ_IN.Auto_Start_Seq, FILL_STT_SEQ4 => "MASTER_FILL_DATA".FILL_STATION_4[4].FILL_SEQ_IN.Auto_Start_Seq, FILL_STT_SEQ5 => "MASTER_FILL_DATA".FILL_STATION_4[5].FILL_SEQ_IN.Auto_Start_Seq, FILL_STT_SEQ6 => "MASTER_FILL_DATA".FILL_STATION_4[6].FILL_SEQ_IN.Auto_Start_Seq, FILLING_SEQ_DONE => "Seq_Lifttable_done", ALL_STATION_DISABLED => %DB504.DBX37.0)
   END_RUNG
   // the same network as SCL:
   IF "AlwaysTRUE" THEN
       #FILLING_STATION4(CYCLE_START := "S4_CYCLE_START",   // "FILLING_FB"
                         CYCLE_RESET := "S4_CYCLE_RESET",
                         CYL_STOPPER := "S4_STOPPER_SENSOR",
                         CYL_SENSOR1 := "S4_SENSOR_CYL1",
                         CYL_SENSOR2 := "S4_SENSOR_CYL2",
                         CYL_SENSOR3 := "S4_SENSOR_CYL3",
                         CYL_SENSOR4 := "S4_SENSOR_CYL4",
                         CYL_SENSOR5 := "S4_SENSOR_CYL5",
                         CYL_SENSOR6 := "S4_SENSOR_CYL6",
                         "DOWN CONVEYOR" := "S4_DOWN_CONVEYOR",
                         "SENSING TIME" := "keypad_logic_DB"."SENSI NG_TIME",
                         ENABLE_CYLINDER := "MASTER_SETUP_DB".S4_Enabled_Station,
                         ENABLED_CYLINDER := "MASTER_SETUP_DB".Enabled_Station_S4,
                         GUN_DELAY_TIME := 2,
                         FILL_SEQ_STARTED := #FILL_SEQ_STARTED,
                         FILLING_DONE := #FILLING_DONE,
                         STOPPER => "S4_STOPPER_OP",
                         "LIFT TABLE1" => "S4_LIFT_CYL1",
                         "LIFT TABLE2" => "S4_LIFT_CYL2",
                         "LIFT TABLE3" => "S4_LIFT_CYL3",
                         "LIFT TABLE4" => "S4_LIFT_CYL4",
                         "LIFT TABLE5" => "S4_LIFT_CYL5",
                         "LIFT TABLE6" => "S4_LIFT_CYL6",
                         FILL_STT_SEQ1 => "MASTER_FILL_DATA".FILL_STATION_4[1].FILL_SEQ_IN.Auto_Start_Seq,
                         FILL_STT_SEQ2 => "MASTER_FILL_DATA".FILL_STATION_4[2].FILL_SEQ_IN.Auto_Start_Seq,
                         FILL_STT_SEQ3 => "MASTER_FILL_DATA".FILL_STATION_4[3].FILL_SEQ_IN.Auto_Start_Seq,
                         FILL_STT_SEQ4 => "MASTER_FILL_DATA".FILL_STATION_4[4].FILL_SEQ_IN.Auto_Start_Seq,
                         FILL_STT_SEQ5 => "MASTER_FILL_DATA".FILL_STATION_4[5].FILL_SEQ_IN.Auto_Start_Seq,
                         FILL_STT_SEQ6 => "MASTER_FILL_DATA".FILL_STATION_4[6].FILL_SEQ_IN.Auto_Start_Seq,
                         FILLING_SEQ_DONE => "Seq_Lifttable_done",
                         ALL_STATION_DISABLED => %DB504.DBX37.0);
   END_IF;
END_REGION

REGION Network 3: Call Filling Line-1 Station-1 FB
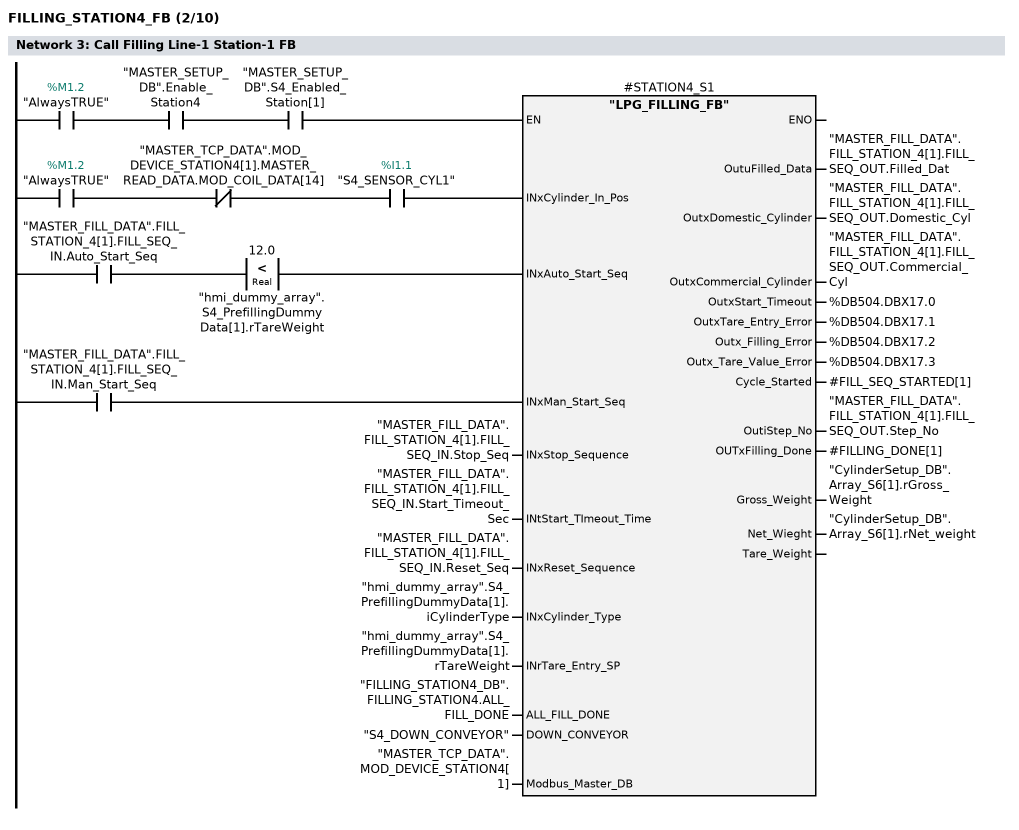
   RUNG wire#powerrail
      Contact( "AlwaysTRUE" )
      Contact( "MASTER_SETUP_DB".Enable_Station4 )
      Contact( "MASTER_SETUP_DB".S4_Enabled_Station[1] )
      #STATION4_S1(INxCylinder_In_Pos := wire#w1, INxAuto_Start_Seq := wire#w2, INxMan_Start_Seq := wire#w3, INxStop_Sequence := "MASTER_FILL_DATA".FILL_STATION_4[1].FILL_SEQ_IN.Stop_Seq, INtStart_TImeout_Time := "MASTER_FILL_DATA".FILL_STATION_4[1].FILL_SEQ_IN.Start_Timeout_Sec, INxReset_Sequence := "MASTER_FILL_DATA".FILL_STATION_4[1].FILL_SEQ_IN.Reset_Seq, INxCylinder_Type := "hmi_dummy_array".S4_PrefillingDummyData[1].iCylinderType, INrTare_Entry_SP := "hmi_dummy_array".S4_PrefillingDummyData[1].rTareWeight, ALL_FILL_DONE := "FILLING_STATION4_DB".FILLING_STATION4.ALL_FILL_DONE, DOWN_CONVEYOR := "S4_DOWN_CONVEYOR", Modbus_Master_DB := "MASTER_TCP_DATA".MOD_DEVICE_STATION4[1], OutuFilled_Data => "MASTER_FILL_DATA".FILL_STATION_4[1].FILL_SEQ_OUT.Filled_Dat, OutxDomestic_Cylinder => "MASTER_FILL_DATA".FILL_STATION_4[1].FILL_SEQ_OUT.Domestic_Cyl, OutxCommercial_Cylinder => "MASTER_FILL_DATA".FILL_STATION_4[1].FILL_SEQ_OUT.Commercial_Cyl, OutxStart_Timeout => %DB504.DBX17.0, OutxTare_Entry_Error => %DB504.DBX17.1, Outx_Filling_Error => %DB504.DBX17.2, Outx_Tare_Value_Error => %DB504.DBX17.3, Cycle_Started => #FILL_SEQ_STARTED[1], OutiStep_No => "MASTER_FILL_DATA".FILL_STATION_4[1].FILL_SEQ_OUT.Step_No, OUTxFilling_Done => #FILLING_DONE[1], Gross_Weight => "CylinderSetup_DB".Array_S6[1].rGross_Weight, Net_Wieght => "CylinderSetup_DB".Array_S6[1].rNet_weight, Tare_Weight =>)
   END_RUNG
   RUNG wire#powerrail
      Contact( "AlwaysTRUE" )
      I_Contact( "MASTER_TCP_DATA".MOD_DEVICE_STATION4[1].MASTER_READ_DATA.MOD_COIL_DATA[14] )
      Contact( "S4_SENSOR_CYL1" )
   END_RUNG wire#w1
   RUNG wire#powerrail
      Contact( "MASTER_FILL_DATA".FILL_STATION_4[1].FILL_SEQ_IN.Auto_Start_Seq )
      { S7_Templates := "SrcType := Real" } LT_Contact(in1 := 12.0, in2 := "hmi_dummy_array".S4_PrefillingDummyData[1].rTareWeight)
   END_RUNG wire#w2
   RUNG wire#powerrail
      Contact( "MASTER_FILL_DATA".FILL_STATION_4[1].FILL_SEQ_IN.Man_Start_Seq )
   END_RUNG wire#w3
   // the same network as SCL:
   IF "AlwaysTRUE" AND "MASTER_SETUP_DB".Enable_Station4 AND "MASTER_SETUP_DB".S4_Enabled_Station[1] THEN
       #STATION4_S1(INxCylinder_In_Pos := "AlwaysTRUE" AND NOT "MASTER_TCP_DATA".MOD_DEVICE_STATION4[1].MASTER_READ_DATA.MOD_COIL_DATA[14] AND "S4_SENSOR_CYL1",   // "LPG_FILLING_FB"
                    INxAuto_Start_Seq := "MASTER_FILL_DATA".FILL_STATION_4[1].FILL_SEQ_IN.Auto_Start_Seq AND (12.0 < "hmi_dummy_array".S4_PrefillingDummyData[1].rTareWeight),
                    INxMan_Start_Seq := "MASTER_FILL_DATA".FILL_STATION_4[1].FILL_SEQ_IN.Man_Start_Seq,
                    INxStop_Sequence := "MASTER_FILL_DATA".FILL_STATION_4[1].FILL_SEQ_IN.Stop_Seq,
                    INtStart_TImeout_Time := "MASTER_FILL_DATA".FILL_STATION_4[1].FILL_SEQ_IN.Start_Timeout_Sec,
                    INxReset_Sequence := "MASTER_FILL_DATA".FILL_STATION_4[1].FILL_SEQ_IN.Reset_Seq,
                    INxCylinder_Type := "hmi_dummy_array".S4_PrefillingDummyData[1].iCylinderType,
                    INrTare_Entry_SP := "hmi_dummy_array".S4_PrefillingDummyData[1].rTareWeight,
                    ALL_FILL_DONE := "FILLING_STATION4_DB".FILLING_STATION4.ALL_FILL_DONE,
                    DOWN_CONVEYOR := "S4_DOWN_CONVEYOR",
                    Modbus_Master_DB := "MASTER_TCP_DATA".MOD_DEVICE_STATION4[1],
                    OutuFilled_Data => "MASTER_FILL_DATA".FILL_STATION_4[1].FILL_SEQ_OUT.Filled_Dat,
                    OutxDomestic_Cylinder => "MASTER_FILL_DATA".FILL_STATION_4[1].FILL_SEQ_OUT.Domestic_Cyl,
                    OutxCommercial_Cylinder => "MASTER_FILL_DATA".FILL_STATION_4[1].FILL_SEQ_OUT.Commercial_Cyl,
                    OutxStart_Timeout => %DB504.DBX17.0,
                    OutxTare_Entry_Error => %DB504.DBX17.1,
                    Outx_Filling_Error => %DB504.DBX17.2,
                    Outx_Tare_Value_Error => %DB504.DBX17.3,
                    Cycle_Started => #FILL_SEQ_STARTED[1],
                    OutiStep_No => "MASTER_FILL_DATA".FILL_STATION_4[1].FILL_SEQ_OUT.Step_No,
                    OUTxFilling_Done => #FILLING_DONE[1],
                    Gross_Weight => "CylinderSetup_DB".Array_S6[1].rGross_Weight,
                    Net_Wieght => "CylinderSetup_DB".Array_S6[1].rNet_weight);
   END_IF;
END_REGION

REGION Network 4: Call Filling Line-1 Station-2 FB
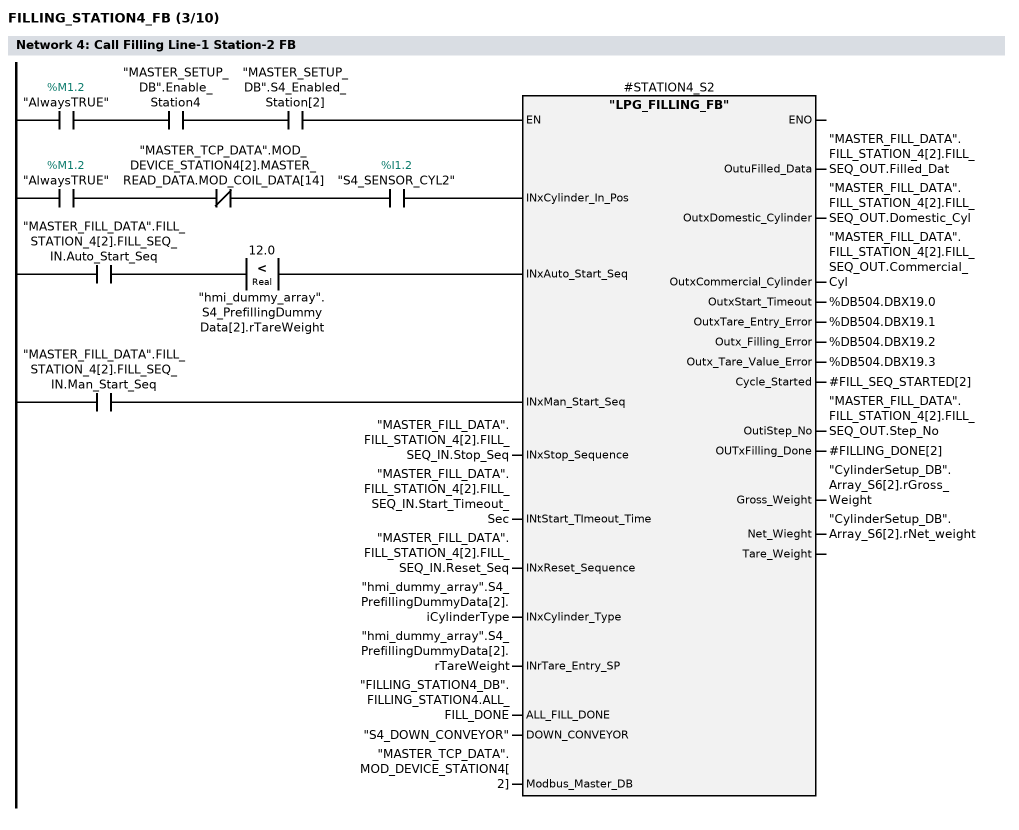
   RUNG wire#powerrail
      Contact( "AlwaysTRUE" )
      Contact( "MASTER_SETUP_DB".Enable_Station4 )
      Contact( "MASTER_SETUP_DB".S4_Enabled_Station[2] )
      #STATION4_S2(INxCylinder_In_Pos := wire#w1, INxAuto_Start_Seq := wire#w2, INxMan_Start_Seq := wire#w3, INxStop_Sequence := "MASTER_FILL_DATA".FILL_STATION_4[2].FILL_SEQ_IN.Stop_Seq, INtStart_TImeout_Time := "MASTER_FILL_DATA".FILL_STATION_4[2].FILL_SEQ_IN.Start_Timeout_Sec, INxReset_Sequence := "MASTER_FILL_DATA".FILL_STATION_4[2].FILL_SEQ_IN.Reset_Seq, INxCylinder_Type := "hmi_dummy_array".S4_PrefillingDummyData[2].iCylinderType, INrTare_Entry_SP := "hmi_dummy_array".S4_PrefillingDummyData[2].rTareWeight, ALL_FILL_DONE := "FILLING_STATION4_DB".FILLING_STATION4.ALL_FILL_DONE, DOWN_CONVEYOR := "S4_DOWN_CONVEYOR", Modbus_Master_DB := "MASTER_TCP_DATA".MOD_DEVICE_STATION4[2], OutuFilled_Data => "MASTER_FILL_DATA".FILL_STATION_4[2].FILL_SEQ_OUT.Filled_Dat, OutxDomestic_Cylinder => "MASTER_FILL_DATA".FILL_STATION_4[2].FILL_SEQ_OUT.Domestic_Cyl, OutxCommercial_Cylinder => "MASTER_FILL_DATA".FILL_STATION_4[2].FILL_SEQ_OUT.Commercial_Cyl, OutxStart_Timeout => %DB504.DBX19.0, OutxTare_Entry_Error => %DB504.DBX19.1, Outx_Filling_Error => %DB504.DBX19.2, Outx_Tare_Value_Error => %DB504.DBX19.3, Cycle_Started => #FILL_SEQ_STARTED[2], OutiStep_No => "MASTER_FILL_DATA".FILL_STATION_4[2].FILL_SEQ_OUT.Step_No, OUTxFilling_Done => #FILLING_DONE[2], Gross_Weight => "CylinderSetup_DB".Array_S6[2].rGross_Weight, Net_Wieght => "CylinderSetup_DB".Array_S6[2].rNet_weight, Tare_Weight =>)
   END_RUNG
   RUNG wire#powerrail
      Contact( "AlwaysTRUE" )
      I_Contact( "MASTER_TCP_DATA".MOD_DEVICE_STATION4[2].MASTER_READ_DATA.MOD_COIL_DATA[14] )
      Contact( "S4_SENSOR_CYL2" )
   END_RUNG wire#w1
   RUNG wire#powerrail
      Contact( "MASTER_FILL_DATA".FILL_STATION_4[2].FILL_SEQ_IN.Auto_Start_Seq )
      { S7_Templates := "SrcType := Real" } LT_Contact(in1 := 12.0, in2 := "hmi_dummy_array".S4_PrefillingDummyData[2].rTareWeight)
   END_RUNG wire#w2
   RUNG wire#powerrail
      Contact( "MASTER_FILL_DATA".FILL_STATION_4[2].FILL_SEQ_IN.Man_Start_Seq )
   END_RUNG wire#w3
   // the same network as SCL:
   IF "AlwaysTRUE" AND "MASTER_SETUP_DB".Enable_Station4 AND "MASTER_SETUP_DB".S4_Enabled_Station[2] THEN
       #STATION4_S2(INxCylinder_In_Pos := "AlwaysTRUE" AND NOT "MASTER_TCP_DATA".MOD_DEVICE_STATION4[2].MASTER_READ_DATA.MOD_COIL_DATA[14] AND "S4_SENSOR_CYL2",   // "LPG_FILLING_FB"
                    INxAuto_Start_Seq := "MASTER_FILL_DATA".FILL_STATION_4[2].FILL_SEQ_IN.Auto_Start_Seq AND (12.0 < "hmi_dummy_array".S4_PrefillingDummyData[2].rTareWeight),
                    INxMan_Start_Seq := "MASTER_FILL_DATA".FILL_STATION_4[2].FILL_SEQ_IN.Man_Start_Seq,
                    INxStop_Sequence := "MASTER_FILL_DATA".FILL_STATION_4[2].FILL_SEQ_IN.Stop_Seq,
                    INtStart_TImeout_Time := "MASTER_FILL_DATA".FILL_STATION_4[2].FILL_SEQ_IN.Start_Timeout_Sec,
                    INxReset_Sequence := "MASTER_FILL_DATA".FILL_STATION_4[2].FILL_SEQ_IN.Reset_Seq,
                    INxCylinder_Type := "hmi_dummy_array".S4_PrefillingDummyData[2].iCylinderType,
                    INrTare_Entry_SP := "hmi_dummy_array".S4_PrefillingDummyData[2].rTareWeight,
                    ALL_FILL_DONE := "FILLING_STATION4_DB".FILLING_STATION4.ALL_FILL_DONE,
                    DOWN_CONVEYOR := "S4_DOWN_CONVEYOR",
                    Modbus_Master_DB := "MASTER_TCP_DATA".MOD_DEVICE_STATION4[2],
                    OutuFilled_Data => "MASTER_FILL_DATA".FILL_STATION_4[2].FILL_SEQ_OUT.Filled_Dat,
                    OutxDomestic_Cylinder => "MASTER_FILL_DATA".FILL_STATION_4[2].FILL_SEQ_OUT.Domestic_Cyl,
                    OutxCommercial_Cylinder => "MASTER_FILL_DATA".FILL_STATION_4[2].FILL_SEQ_OUT.Commercial_Cyl,
                    OutxStart_Timeout => %DB504.DBX19.0,
                    OutxTare_Entry_Error => %DB504.DBX19.1,
                    Outx_Filling_Error => %DB504.DBX19.2,
                    Outx_Tare_Value_Error => %DB504.DBX19.3,
                    Cycle_Started => #FILL_SEQ_STARTED[2],
                    OutiStep_No => "MASTER_FILL_DATA".FILL_STATION_4[2].FILL_SEQ_OUT.Step_No,
                    OUTxFilling_Done => #FILLING_DONE[2],
                    Gross_Weight => "CylinderSetup_DB".Array_S6[2].rGross_Weight,
                    Net_Wieght => "CylinderSetup_DB".Array_S6[2].rNet_weight);
   END_IF;
END_REGION

REGION Network 5: Call Filling Line-1 Station-3 FB
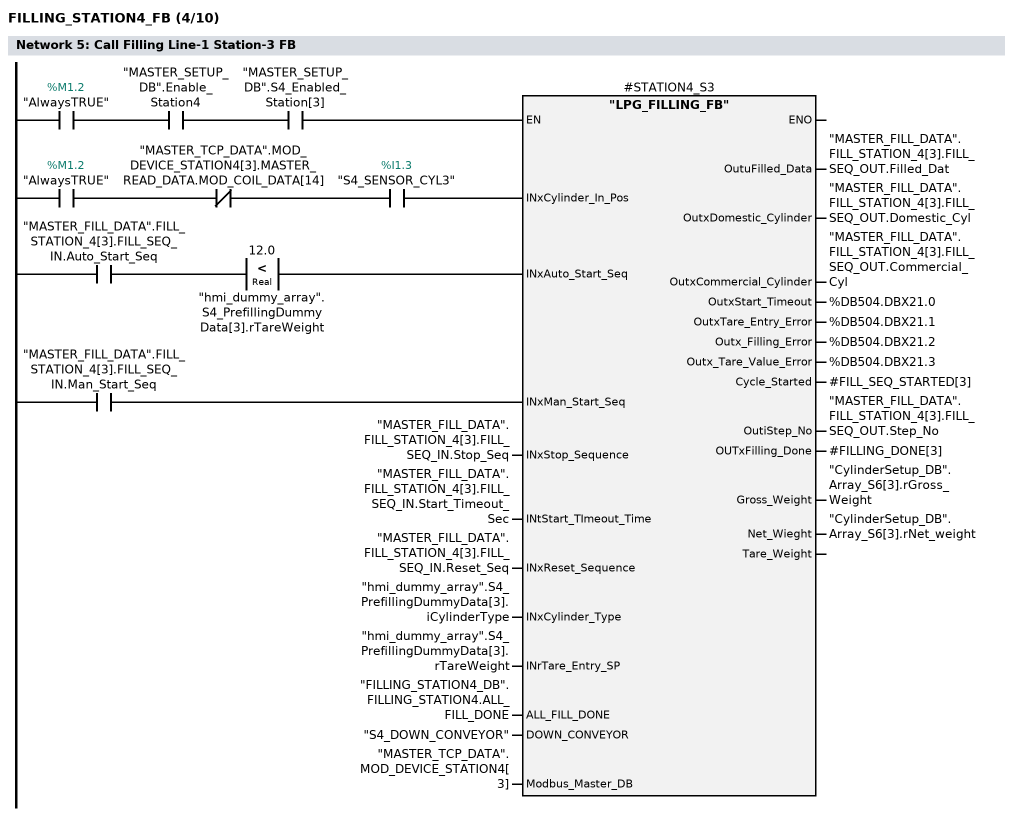
   RUNG wire#powerrail
      Contact( "AlwaysTRUE" )
      Contact( "MASTER_SETUP_DB".Enable_Station4 )
      Contact( "MASTER_SETUP_DB".S4_Enabled_Station[3] )
      #STATION4_S3(INxCylinder_In_Pos := wire#w1, INxAuto_Start_Seq := wire#w2, INxMan_Start_Seq := wire#w3, INxStop_Sequence := "MASTER_FILL_DATA".FILL_STATION_4[3].FILL_SEQ_IN.Stop_Seq, INtStart_TImeout_Time := "MASTER_FILL_DATA".FILL_STATION_4[3].FILL_SEQ_IN.Start_Timeout_Sec, INxReset_Sequence := "MASTER_FILL_DATA".FILL_STATION_4[3].FILL_SEQ_IN.Reset_Seq, INxCylinder_Type := "hmi_dummy_array".S4_PrefillingDummyData[3].iCylinderType, INrTare_Entry_SP := "hmi_dummy_array".S4_PrefillingDummyData[3].rTareWeight, ALL_FILL_DONE := "FILLING_STATION4_DB".FILLING_STATION4.ALL_FILL_DONE, DOWN_CONVEYOR := "S4_DOWN_CONVEYOR", Modbus_Master_DB := "MASTER_TCP_DATA".MOD_DEVICE_STATION4[3], OutuFilled_Data => "MASTER_FILL_DATA".FILL_STATION_4[3].FILL_SEQ_OUT.Filled_Dat, OutxDomestic_Cylinder => "MASTER_FILL_DATA".FILL_STATION_4[3].FILL_SEQ_OUT.Domestic_Cyl, OutxCommercial_Cylinder => "MASTER_FILL_DATA".FILL_STATION_4[3].FILL_SEQ_OUT.Commercial_Cyl, OutxStart_Timeout => %DB504.DBX21.0, OutxTare_Entry_Error => %DB504.DBX21.1, Outx_Filling_Error => %DB504.DBX21.2, Outx_Tare_Value_Error => %DB504.DBX21.3, Cycle_Started => #FILL_SEQ_STARTED[3], OutiStep_No => "MASTER_FILL_DATA".FILL_STATION_4[3].FILL_SEQ_OUT.Step_No, OUTxFilling_Done => #FILLING_DONE[3], Gross_Weight => "CylinderSetup_DB".Array_S6[3].rGross_Weight, Net_Wieght => "CylinderSetup_DB".Array_S6[3].rNet_weight, Tare_Weight =>)
   END_RUNG
   RUNG wire#powerrail
      Contact( "AlwaysTRUE" )
      I_Contact( "MASTER_TCP_DATA".MOD_DEVICE_STATION4[3].MASTER_READ_DATA.MOD_COIL_DATA[14] )
      Contact( "S4_SENSOR_CYL3" )
   END_RUNG wire#w1
   RUNG wire#powerrail
      Contact( "MASTER_FILL_DATA".FILL_STATION_4[3].FILL_SEQ_IN.Auto_Start_Seq )
      { S7_Templates := "SrcType := Real" } LT_Contact(in1 := 12.0, in2 := "hmi_dummy_array".S4_PrefillingDummyData[3].rTareWeight)
   END_RUNG wire#w2
   RUNG wire#powerrail
      Contact( "MASTER_FILL_DATA".FILL_STATION_4[3].FILL_SEQ_IN.Man_Start_Seq )
   END_RUNG wire#w3
   // the same network as SCL:
   IF "AlwaysTRUE" AND "MASTER_SETUP_DB".Enable_Station4 AND "MASTER_SETUP_DB".S4_Enabled_Station[3] THEN
       #STATION4_S3(INxCylinder_In_Pos := "AlwaysTRUE" AND NOT "MASTER_TCP_DATA".MOD_DEVICE_STATION4[3].MASTER_READ_DATA.MOD_COIL_DATA[14] AND "S4_SENSOR_CYL3",   // "LPG_FILLING_FB"
                    INxAuto_Start_Seq := "MASTER_FILL_DATA".FILL_STATION_4[3].FILL_SEQ_IN.Auto_Start_Seq AND (12.0 < "hmi_dummy_array".S4_PrefillingDummyData[3].rTareWeight),
                    INxMan_Start_Seq := "MASTER_FILL_DATA".FILL_STATION_4[3].FILL_SEQ_IN.Man_Start_Seq,
                    INxStop_Sequence := "MASTER_FILL_DATA".FILL_STATION_4[3].FILL_SEQ_IN.Stop_Seq,
                    INtStart_TImeout_Time := "MASTER_FILL_DATA".FILL_STATION_4[3].FILL_SEQ_IN.Start_Timeout_Sec,
                    INxReset_Sequence := "MASTER_FILL_DATA".FILL_STATION_4[3].FILL_SEQ_IN.Reset_Seq,
                    INxCylinder_Type := "hmi_dummy_array".S4_PrefillingDummyData[3].iCylinderType,
                    INrTare_Entry_SP := "hmi_dummy_array".S4_PrefillingDummyData[3].rTareWeight,
                    ALL_FILL_DONE := "FILLING_STATION4_DB".FILLING_STATION4.ALL_FILL_DONE,
                    DOWN_CONVEYOR := "S4_DOWN_CONVEYOR",
                    Modbus_Master_DB := "MASTER_TCP_DATA".MOD_DEVICE_STATION4[3],
                    OutuFilled_Data => "MASTER_FILL_DATA".FILL_STATION_4[3].FILL_SEQ_OUT.Filled_Dat,
                    OutxDomestic_Cylinder => "MASTER_FILL_DATA".FILL_STATION_4[3].FILL_SEQ_OUT.Domestic_Cyl,
                    OutxCommercial_Cylinder => "MASTER_FILL_DATA".FILL_STATION_4[3].FILL_SEQ_OUT.Commercial_Cyl,
                    OutxStart_Timeout => %DB504.DBX21.0,
                    OutxTare_Entry_Error => %DB504.DBX21.1,
                    Outx_Filling_Error => %DB504.DBX21.2,
                    Outx_Tare_Value_Error => %DB504.DBX21.3,
                    Cycle_Started => #FILL_SEQ_STARTED[3],
                    OutiStep_No => "MASTER_FILL_DATA".FILL_STATION_4[3].FILL_SEQ_OUT.Step_No,
                    OUTxFilling_Done => #FILLING_DONE[3],
                    Gross_Weight => "CylinderSetup_DB".Array_S6[3].rGross_Weight,
                    Net_Wieght => "CylinderSetup_DB".Array_S6[3].rNet_weight);
   END_IF;
END_REGION

REGION Network 6: Call Filling Line-1 Station-4 FB
